# B&R Automation Studio project OpcUaSample410_BrbLibUa103 (part 6)

#### BrbStringPadLeft.c - Füllt einen String auf der linken Seite mit einem Füllzeichen auf eine bestimme Länge
```c
/********************************************************************
 * COPYRIGHT -- Bernecker + Rainer
 ********************************************************************
 * Library: BrbLib
 * File: BrbStringPadLeft.c
 * Author: niedermeierr
 * Created: June 11, 2013
 ********************************************************************
 * Implementation of library BrbLib
 ********************************************************************/

#include <bur/plctypes.h>
#ifdef __cplusplus
	extern "C"
	{
#endif

#include "BrbLib.h"
#include <string.h>

#ifdef __cplusplus
	};
#endif

// NOLINTBEGIN(readability-*, bugprone-easily-swappable-parameters, clang-diagnostic-invalid-utf8, clang-diagnostic-invalid-source-encoding, clang-diagnostic-pointer-arith, clang-diagnostic-strict-prototypes, hicpp-uppercase-literal-suffix, cppcoreguidelines-*, performance-*)

/* Füllt einen String auf der linken Seite mit einem Füllzeichen auf eine bestimme Länge */
plcbit BrbStringPadLeft(plcstring* pText, plcstring* pFillChar, unsigned long nLen)
{
	BOOL bResult = 0;
	UDINT nTextLen = strlen(pText);
	DINT nFillLen = (DINT)nLen - (DINT)nTextLen;
	USINT* pChar = (USINT*)pText;
	if(nFillLen > 0)
	{
		// Text nach rechts schieben
		memmove(pText+nFillLen, pText, nTextLen+1);
		// Füllzeichen einsetzen
		while(pChar < (USINT*)(pText+nFillLen))
		{
			*pChar = (USINT)*pFillChar;
			pChar++;
		}
		bResult = 1;
	}
	return bResult;
}

// NOLINTEND(readability-*, bugprone-easily-swappable-parameters, clang-diagnostic-invalid-utf8, clang-diagnostic-invalid-source-encoding, clang-diagnostic-pointer-arith, clang-diagnostic-strict-prototypes, hicpp-uppercase-literal-suffix, cppcoreguidelines-*, performance-*)
```

#### BrbStringPadRight.c - Füllt einen String auf der rechten Seite mit einem Füllzeichen auf eine bestimme Länge
```c
/********************************************************************
 * COPYRIGHT -- Bernecker + Rainer
 ********************************************************************
 * Library: BrbLib
 * File: BrbStringPadRight.c
 * Author: niedermeierr
 * Created: June 11, 2013
 ********************************************************************
 * Implementation of library BrbLib
 ********************************************************************/

#include <bur/plctypes.h>
#ifdef __cplusplus
	extern "C"
	{
#endif

#include "BrbLib.h"
#include <string.h>

#ifdef __cplusplus
	};
#endif

// NOLINTBEGIN(readability-*, bugprone-easily-swappable-parameters, clang-diagnostic-invalid-utf8, clang-diagnostic-invalid-source-encoding, clang-diagnostic-pointer-arith, clang-diagnostic-strict-prototypes, hicpp-uppercase-literal-suffix, cppcoreguidelines-*, performance-*)

/* Füllt einen String auf der rechten Seite mit einem Füllzeichen auf eine bestimme Länge */
plcbit BrbStringPadRight(plcstring* pText, plcstring* pFillChar, unsigned long nLen)
{
	BOOL bResult = 0;
	UDINT nTextLen = strlen(pText);
	DINT nFillLen = (DINT)nLen - (DINT)nTextLen;
	USINT* pChar = (USINT*)pText + nTextLen;
	if(nFillLen > 0)
	{
		// Füllzeichen einsetzen
		while(pChar < (USINT*)(pText+nLen))
		{
			*pChar = (USINT)*pFillChar;
			pChar++;
		}
		bResult = 1;
	}
	// Terminierung
	*pChar = 0;
	return bResult;
}

// NOLINTEND(readability-*, bugprone-easily-swappable-parameters, clang-diagnostic-invalid-utf8, clang-diagnostic-invalid-source-encoding, clang-diagnostic-pointer-arith, clang-diagnostic-strict-prototypes, hicpp-uppercase-literal-suffix, cppcoreguidelines-*, performance-*)
```

#### BrbStringTrimLeft.c - Schneidet eine Zeichenfolge auf der linken Seite eines Textes heraus
```c
/********************************************************************
 * COPYRIGHT -- Bernecker + Rainer
 ********************************************************************
 * Library: BrbLib
 * File: BrbStringTrimLeft.c
 * Author: niedermeierr
 * Created: December 03, 2013
 ********************************************************************
 * Implementation of library BrbLib
 ********************************************************************/

#include <bur/plctypes.h>
#ifdef __cplusplus
	extern "C"
	{
#endif

#include "BrbLib.h"
#include <string.h>

#ifdef __cplusplus
	};
#endif

// NOLINTBEGIN(readability-*, bugprone-easily-swappable-parameters, clang-diagnostic-invalid-utf8, clang-diagnostic-invalid-source-encoding, clang-diagnostic-pointer-arith, clang-diagnostic-strict-prototypes, hicpp-uppercase-literal-suffix, cppcoreguidelines-*, performance-*)

/* Schneidet eine Zeichenfolge auf der linken Seite eines Textes heraus */
plcbit BrbStringTrimLeft(plcstring* pText, plcstring* pTrim)
{
	BOOL bResult = 0;
	UDINT nTrimLen = strlen(pTrim);
	BOOL bLeave = 0;
	do
	{
		if(BrbStringStartsWith(pText, pTrim) == 1)
		{
			BrbStringCut(pText, 0, nTrimLen, 0);
			bResult = 1;
		}
		else
		{
			bLeave = 1;
		}
	} while(bLeave == 0);
	return bResult;
}

// NOLINTEND(readability-*, bugprone-easily-swappable-parameters, clang-diagnostic-invalid-utf8, clang-diagnostic-invalid-source-encoding, clang-diagnostic-pointer-arith, clang-diagnostic-strict-prototypes, hicpp-uppercase-literal-suffix, cppcoreguidelines-*, performance-*)
```

#### BrbStringTrimRight.c - Schneidet eine Zeichenfolge auf der rechten Seite eines Textes heraus
```c
/********************************************************************
 * COPYRIGHT -- Bernecker + Rainer
 ********************************************************************
 * Library: BrbLib
 * File: BrbStringTrimRight.c
 * Author: niedermeierr
 * Created: December 03, 2013
 ********************************************************************
 * Implementation of library BrbLib
 ********************************************************************/

#include <bur/plctypes.h>
#ifdef __cplusplus
	extern "C"
	{
#endif

#include "BrbLib.h"
#include <string.h>

#ifdef __cplusplus
	};
#endif

// NOLINTBEGIN(readability-*, bugprone-easily-swappable-parameters, clang-diagnostic-invalid-utf8, clang-diagnostic-invalid-source-encoding, clang-diagnostic-pointer-arith, clang-diagnostic-strict-prototypes, hicpp-uppercase-literal-suffix, cppcoreguidelines-*, performance-*)

/* Schneidet eine Zeichenfolge auf der rechten Seite eines Textes heraus */
plcbit BrbStringTrimRight(plcstring* pText, plcstring* pTrim)
{
	BOOL bResult = 0;
	UDINT nTrimLen = strlen(pTrim);
	BOOL bLeave = 0;
	do
	{
		if(BrbStringEndsWith(pText, pTrim) == 1)
		{
			UDINT nTextLen = strlen(pText);
			BrbStringCut(pText, nTextLen-nTrimLen, nTrimLen, 0);
			bResult = 1;
		}
		else
		{
			bLeave = 1;
		}
	} while(bLeave == 0);
	return bResult;
}

// NOLINTEND(readability-*, bugprone-easily-swappable-parameters, clang-diagnostic-invalid-utf8, clang-diagnostic-invalid-source-encoding, clang-diagnostic-pointer-arith, clang-diagnostic-strict-prototypes, hicpp-uppercase-literal-suffix, cppcoreguidelines-*, performance-*)
```

#### BrbStringSplit.c - Spaltet einen Text in mehrere String aufgrund eines Trennzeichens
```c
/********************************************************************
 * COPYRIGHT -- Bernecker + Rainer
 ********************************************************************
 * Library: BrbLib
 * File: BrbStringSplit.c
 * Author: niedermeierr
 * Created: June 17, 2013
 ********************************************************************
 * Implementation of library BrbLib
 ********************************************************************/

#include <bur/plctypes.h>
#ifdef __cplusplus
	extern "C"
	{
#endif

#include "BrbLib.h"
#include <string.h>

#ifdef __cplusplus
	};
#endif

// NOLINTBEGIN(readability-*, bugprone-easily-swappable-parameters, clang-diagnostic-invalid-utf8, clang-diagnostic-invalid-source-encoding, clang-diagnostic-pointer-arith, clang-diagnostic-strict-prototypes, hicpp-uppercase-literal-suffix, cppcoreguidelines-*, performance-*)

/* Spaltet einen Text in mehrere Strings aufgrund eines Trennzeichens */
unsigned long BrbStringSplit(plcstring* pText, plcstring* pSep, unsigned long pSplitArray, unsigned long nArrayIndexMax, unsigned long nEntrySize)
{
	if(nEntrySize <= 1)
	{
		// String-Grösse zu klein
		return 0;
	}
	UDINT nResult = 0;
	UDINT nLenText = strlen(pText);
	UDINT nLenSep = strlen(pSep);
	// Der Einfachkeit halber wird das Array in einer MemList verwaltet
	BrbMemListManagement_Typ ListMan;
	ListMan.pList = pSplitArray;
	ListMan.nIndexMax = nArrayIndexMax;
	ListMan.nEntryLength = nEntrySize;
	BrbMemListClear(&ListMan);
	// Text von vorne nach hinten nach Trennzeichen durchsuchen
	STRING* pEntryTextStart = pText;
	STRING* pEntryTextEnd = 0;
	UDINT nCharIndex = 0;
	do
	{
		// Trennzeichen vergleichen
		if((memcmp((pText + nCharIndex), pSep, nLenSep) == 0) || nCharIndex == nLenText-1)
		{
			// Trennzeichen gefunden -> Splittext holen und in Array eintragen
			if(nCharIndex == nLenText-1)
			{
				// Kein Trennzeichen am Ende
				pEntryTextEnd = pText + nCharIndex + 1;
			}
			else
			{
				pEntryTextEnd = pText + nCharIndex;
			}
			STRING sEntryText[nEntrySize];
			memset(sEntryText, 0, sizeof(sEntryText));
			DINT nNeededEntrySize = (DINT)pEntryTextEnd - (DINT)pEntryTextStart + 1;
			if((DINT)nEntrySize < nNeededEntrySize)
			{
				pEntryTextEnd = pEntryTextStart + nEntrySize - 1;
			}
			BrbStringGetSubTextByAdr(pEntryTextStart, pEntryTextEnd, sEntryText);
			if(strlen(sEntryText) > 0 && strcmp(sEntryText, pSep) != 0)
			{
				BrbMemListIn(&ListMan, ListMan.nEntryCount, (UDINT)&sEntryText);
				nResult += 1;
			}
			// Weitermachen mit Text nach Trennzeichen
			nCharIndex += nLenSep;
			pEntryTextStart = pText + nCharIndex;
		}
		else
		{
			nCharIndex += 1;
		}
	} while(nCharIndex<nLenText);
	return nResult;
}

// NOLINTEND(readability-*, bugprone-easily-swappable-parameters, clang-diagnostic-invalid-utf8, clang-diagnostic-invalid-source-encoding, clang-diagnostic-pointer-arith, clang-diagnostic-strict-prototypes, hicpp-uppercase-literal-suffix, cppcoreguidelines-*, performance-*)
```

#### BrbStringSplitEmpty.c - Spaltet einen Text in mehrere String aufgrund eines Trennzeichens
```c
/********************************************************************
 * COPYRIGHT -- Bernecker + Rainer
 ********************************************************************
 * Library: BrbLib
 * File: BrbStringSplitEmpty.c
 * Author: niedermeierr
 * Created: May 17, 2021
 ********************************************************************
 * Implementation of library BrbLib
 ********************************************************************/

#include <bur/plctypes.h>
#ifdef __cplusplus
	extern "C"
	{
#endif

#include "BrbLib.h"
#include <string.h>

#ifdef __cplusplus
	};
#endif

// NOLINTBEGIN(readability-*, bugprone-easily-swappable-parameters, clang-diagnostic-invalid-utf8, clang-diagnostic-invalid-source-encoding, clang-diagnostic-pointer-arith, clang-diagnostic-strict-prototypes, hicpp-uppercase-literal-suffix, cppcoreguidelines-*, performance-*)

/* Spaltet einen Text in mehrere Strings aufgrund eines Trennzeichens (inkl. Leer-Strings) */
unsigned long BrbStringSplitEmpty(plcstring* pText, plcstring* pSep, unsigned long pSplitArray, unsigned long nArrayIndexMax, unsigned long nEntrySize)
{
	if(nEntrySize <= 1)
	{
		// String-Grösse zu klein
		return 0;
	}
	UDINT nResult = 0;
	UDINT nLenText = strlen(pText);
	UDINT nLenSep = strlen(pSep);
	// Der Einfachkeit halber wird das Array in einer MemList verwaltet
	BrbMemListManagement_Typ ListMan;
	ListMan.pList = pSplitArray;
	ListMan.nIndexMax = nArrayIndexMax;
	ListMan.nEntryLength = nEntrySize;
	BrbMemListClear(&ListMan);
	// Text von vorne nach hinten nach Trennzeichen durchsuchen
	STRING* pEntryTextStart = pText;
	STRING* pEntryTextEnd = 0;
	UDINT nCharIndex = 0;
	do
	{
		// Trennzeichen vergleichen
		if((memcmp((pText + nCharIndex), pSep, nLenSep) == 0) || nCharIndex == nLenText-1)
		{
			// Trennzeichen gefunden -> Splittext holen und in Array eintragen
			if((memcmp((pText + nCharIndex), pSep, nLenSep) != 0) && nCharIndex == nLenText-1)
			{
				// Kein Trennzeichen am Ende
				pEntryTextEnd = pText + nCharIndex + 1;
			}
			else
			{
				pEntryTextEnd = pText + nCharIndex;
			}
			STRING sEntryText[nEntrySize];
			memset(sEntryText, 0, sizeof(sEntryText));
			DINT nNeededEntrySize = (DINT)pEntryTextEnd - (DINT)pEntryTextStart + 1;
			if((DINT)nEntrySize < nNeededEntrySize)
			{
				pEntryTextEnd = pEntryTextStart + nEntrySize - 1;
			}
			BrbStringGetSubTextByAdr(pEntryTextStart, pEntryTextEnd, sEntryText);
			if(strcmp(sEntryText, pSep) == 0)
			{
				memset(sEntryText, 0, sizeof(sEntryText));
			}
			BrbMemListIn(&ListMan, ListMan.nEntryCount, (UDINT)&sEntryText);
			nResult += 1;
			// Weitermachen mit Text nach Trennzeichen
			nCharIndex += nLenSep;
			pEntryTextStart = pText + nCharIndex;
		}
		else
		{
			nCharIndex += 1;
		}
	} while(nCharIndex<nLenText);
	if(pEntryTextEnd != 0)
	{
		if(BrbStringEndsWith(pEntryTextEnd, pSep) == 1)
		{
			// Text endet mit Trennzeichen -> noch einen leeren Eintrag hinzufügen
			STRING sEntryText[nEntrySize];
			memset(sEntryText, 0, sizeof(sEntryText));
			BrbMemListIn(&ListMan, ListMan.nEntryCount, (UDINT)&sEntryText);
			nResult += 1;
		}
	}
	return nResult;
}

// NOLINTEND(readability-*, bugprone-easily-swappable-parameters, clang-diagnostic-invalid-utf8, clang-diagnostic-invalid-source-encoding, clang-diagnostic-pointer-arith, clang-diagnostic-strict-prototypes, hicpp-uppercase-literal-suffix, cppcoreguidelines-*, performance-*)
```

#### BrbStringConvertRealFromExp.c - Konvertiert eine exponentielle Notation in einen Real-Wert
```c
/********************************************************************
 * COPYRIGHT -- Bernecker + Rainer
 ********************************************************************
 * Library: BrbLib
 * File: BrbStringConvertRealFromExp.c
 * Author: niedermeierr
 * Created: December 03, 2013
 ********************************************************************
 * Implementation of library BrbLib
 ********************************************************************/

#include <bur/plctypes.h>
#ifdef __cplusplus
	extern "C"
	{
#endif

#include "BrbLib.h"
#include <string.h>
#include <AnsiCFunc.h>

#ifdef __cplusplus
	};
#endif

// NOLINTBEGIN(readability-*, bugprone-easily-swappable-parameters, clang-diagnostic-invalid-utf8, clang-diagnostic-invalid-source-encoding, clang-diagnostic-pointer-arith, clang-diagnostic-strict-prototypes, hicpp-uppercase-literal-suffix, cppcoreguidelines-*, performance-*)

/* Konvertiert eine exponentielle Notation in einen Real-Wert */
unsigned short BrbStringConvertRealFromExp(plcstring* pValue, plcstring* pResult, unsigned long nResultSize) // NOLINT(readability-function-cognitive-complexity)
{
	memset(pResult, 0, nResultSize);
	UDINT nValueLen = strlen(pValue);
	STRING* pExpStart = BrbStringGetAdrOf(pValue, "e", nValueLen);
	if(pExpStart > pValue)
	{
		// "e" enthalten -> Zahl vor dem "e"
		STRING sReal[50];
		memset(sReal, 0, sizeof(sReal));
		BrbStringGetSubTextByAdr(pValue, pExpStart, sReal); // NOLINT(readability-suspicious-call-argument)
		// Vorzeichen, Anzahl der Vorkomma-Stellen, Stelle des Kommas und Anzahl der Nachkomma-Stellen
		BOOL bMinus = 0;
		// Vorzeichen löschen
		BrbStringTrimLeft(sReal, "+");
		if(BrbStringStartsWith(sReal, "-") == 1)
		{
			bMinus = 1;
			BrbStringTrimLeft(sReal, "-");
		}
		// Führende Nullen löschen
		BrbStringTrimLeft(sReal, "0");

		STRING* pRealDot = BrbStringGetAdrOf(sReal, ".", nValueLen);
		UDINT nIntegerDigits = 0;
		DINT nDotDigit = 0;
		UDINT nFractionDigits = 0;
		if((UDINT)pRealDot >= (UDINT)&sReal)
		{
			// Punkt enthalten
			// Folgende Nullen nach dem Punkt löschen
			BrbStringTrimRight(sReal, "0");
			if(BrbStringEndsWith(sReal, ".") == 1)
			{
				brsstrcat((UDINT)&sReal, (UDINT)&"0");
			}
			UDINT nRealLen = strlen(sReal);
			nIntegerDigits = (UDINT)pRealDot - (UDINT)sReal;
			nDotDigit = (DINT)((UDINT)pRealDot - (UDINT)&sReal);
			nFractionDigits = (UDINT)&sReal + nRealLen - (UDINT)pRealDot - 1;
			// Punkt löschen
			BrbStringReplace(sReal, ".", "");
		}
		else
		{
			// Punkt nicht enthalten
			nIntegerDigits = (UDINT)pExpStart - (UDINT)pValue;
			nDotDigit = -1;
			nFractionDigits = 0;
		}
		brsstrcpy((UDINT)pResult, (UDINT)&sReal);
		UDINT nExpLen = strlen(pExpStart);
		if(nExpLen > 1)
		{
			// Zahl nach dem "e"
			STRING sExp[50];
			memset(sExp, 0, sizeof(sExp));
			BrbStringGetSubTextByLen(pExpStart + 1, nExpLen - 1, sExp);
			DINT nExp = brsatoi((UDINT)&sExp);
			// Vorzeichen des Exponenten
			STRING* pExpMinus = BrbStringGetAdrOf(pExpStart, "-", nExpLen);
			if(pExpMinus > pExpStart && nExp != 0)
			{
				// Exponent ist negativ -> Nullen voranstellen
				UDINT nAddZero = (UDINT)((DINT)abs(nExp) - (DINT)nIntegerDigits) + 1;
				UDINT nCount = 0;
				for(nCount=0; nCount<nAddZero; nCount++)
				{
					BrbStringInsert(pResult, 0, "0");
				}
				// Punkt einfügen
				BrbStringInsert(pResult, 1, ".");
			}
			else
			{
				// Exponent ist positiv
				if((DINT)nFractionDigits <= nExp)
				{
					// Nullen anhängen
					UDINT nAddZero = (UDINT)(nExp - (DINT)nFractionDigits);
					UDINT nCount = 0;
					for(nCount=0; nCount<nAddZero; nCount++)
					{
						brsstrcat((UDINT)pResult, (UDINT)&"0");
					}
				}
				else
				{
					// Punkt einfügen
					if(nDotDigit > -1)
					{
						UDINT nIndex = (UDINT)(nDotDigit + nExp);
						BrbStringInsert(pResult, nIndex, ".");
					}
				}
			}
			// Führende Nullen löschen
			BrbStringTrimLeft(pResult, "0");
			// Null vor dem Punkt wieder einfügen
			if(BrbStringStartsWith(pResult, ".") == 1)
			{
				BrbStringInsert(pResult, 0, "0");
			}
			// Vorzeichen einfügen
			if(bMinus == 1)
			{
				BrbStringInsert(pResult, 0, "-");
			}
		}
	}
	else
	{
		// "e" nicht enthalten
		brsstrcpy((UDINT)pResult, (UDINT)pValue);
		// Vorzeichen löschen
		BrbStringTrimLeft(pResult, "+");
		BOOL bMinus = 0;
		if(BrbStringStartsWith(pResult, "-") == 1)
		{
			bMinus = 1;
			BrbStringTrimLeft(pResult, "-");
		}
		// Führende Nullen löschen
		BrbStringTrimLeft(pResult, "0");
		// Null vor dem Punkt wieder einfügen
		if(BrbStringStartsWith(pResult, ".") == 1)
		{
			BrbStringInsert(pResult, 0, "0");
		}
		// Folgende Nullen nach dem Punkt löschen
		UDINT nLen = strlen(pResult);
		STRING* pDot = BrbStringGetAdrOf(pResult, ".", nLen);
		if(pDot > pResult)
		{
			BrbStringTrimRight(pResult, "0");
			if(BrbStringEndsWith(pResult, ".") == 1)
			{
				brsstrcat((UDINT)pResult, (UDINT)&"0");
			}
		}
		if(strlen(pResult) == 0)
		{
			brsstrcat((UDINT)pResult, (UDINT)&"0.0");
		}
		// Vorzeichen einfügen
		if(bMinus == 1)
		{
			BrbStringInsert(pResult, 0, "-");
		}
	}
	return eBRB_ERR_OK;
}

// NOLINTEND(readability-*, bugprone-easily-swappable-parameters, clang-diagnostic-invalid-utf8, clang-diagnostic-invalid-source-encoding, clang-diagnostic-pointer-arith, clang-diagnostic-strict-prototypes, hicpp-uppercase-literal-suffix, cppcoreguidelines-*, performance-*)
```

#### BrbStringConvertRealToExp.c - Konvertiert einen Real-Wert in eine exponentielle Notation
```c
/********************************************************************
 * COPYRIGHT -- Bernecker + Rainer
 ********************************************************************
 * Library: BrbLib
 * File: BrbStringConvertRealToExp.c
 * Author: niedermeierr
 * Created: December 03, 2013
 ********************************************************************
 * Implementation of library BrbLib
 ********************************************************************/

#include <bur/plctypes.h>
#ifdef __cplusplus
	extern "C"
	{
#endif

#include "BrbLib.h"
#include <string.h>
#include <AnsiCFunc.h>

#ifdef __cplusplus
	};
#endif

// NOLINTBEGIN(readability-*, bugprone-easily-swappable-parameters, clang-diagnostic-invalid-utf8, clang-diagnostic-invalid-source-encoding, clang-diagnostic-pointer-arith, clang-diagnostic-strict-prototypes, hicpp-uppercase-literal-suffix, cppcoreguidelines-*, performance-*)

/* Konvertiert einen Real-Wert in eine exponentielle Notation */
unsigned short BrbStringConvertRealToExp(plcstring* pValue, plcstring* pResult, unsigned long nResultSize) // NOLINT(readability-function-cognitive-complexity)
{
	memset(pResult, 0, nResultSize);
	UDINT nValueLen = strlen(pValue);
	STRING* pExpStart = BrbStringGetAdrOf(pValue, "e", nValueLen);
	if(pExpStart == 0)
	{
		// "e" nicht enthalten
		brsstrcpy((UDINT)pResult, (UDINT)pValue);
		// Vorzeichen löschen
		BrbStringTrimLeft(pResult, "+");
		BOOL bMinus = 0;
		if(BrbStringStartsWith(pResult, "-") == 1)
		{
			bMinus = 1;
			BrbStringTrimLeft(pResult, "-");
		}
		// Führende Nullen löschen
		BrbStringTrimLeft(pResult, "0");
		// Null vor dem Punkt wieder einfügen
		if(BrbStringStartsWith(pResult, ".") == 1)
		{
			BrbStringInsert(pResult, 0, "0");
		}
		else if(brsstrlen((UDINT)pResult) == 0)
		{
			brsstrcat((UDINT)pResult, (UDINT)&"0.0");
		}
		// Folgende Nullen nach dem Punkt löschen
		UDINT nLen = strlen(pResult);
		STRING* pDot = BrbStringGetAdrOf(pResult, ".", nLen);
		if(pDot > pResult)
		{
			BrbStringTrimRight(pResult, "0");
			if(BrbStringEndsWith(pResult, ".") == 1)
			{
				brsstrcat((UDINT)pResult, (UDINT)&"0");
			}
			nLen = strlen(pResult);
			pDot = BrbStringGetAdrOf(pResult, ".", nLen);
		}
		// Vorzeichen des Exponenten feststellen
		BOOL bExpMinus = 0;
		if(BrbStringStartsWith(pResult, "0") == 1)
		{
			// 0.0012345
			// Erstes Zeichen ist "0" -> Exponent negativ
			bExpMinus = 1;
		}
		else
		{
			// 123.45
			// Erstes Zeichen ist keine "0" -> Exponent positiv
			bExpMinus = 0;
		}
		// Exponent feststellen
		DINT nExp = 0;
		if(bExpMinus == 1)
		{
			// Negativer Exponent
			if(pDot > pResult)
			{
				// Punkt enthalten
				nExp = 1;
				USINT* pChar = 0;
				USINT* pEnd =(USINT*)pResult + nLen - 1;
				// Anzahl der Nullen vom Punkt bis zur ersten relevanten Ziffer
				for(pChar=(USINT*)pDot+1; pChar<=pEnd; pChar++)
				{
					if(*pChar == 48)
					{
						nExp += 1;
					}
					else
					{
						break;
					}
				}
				UDINT nDotDigit = (UDINT)pDot - (UDINT)pResult;
				UDINT nCutLen = nDotDigit + (UDINT)nExp;
				// Alle Zeichen bis zur ersten relevanten Ziffer löschen
				BrbStringCut(pResult, 0, nCutLen, 0);
			}
			else
			{
				// Punkt nicht enthalten
				nExp = 0;
			}
		}
		else
		{
			// Positiver Exponent
			if(pDot > pResult)
			{
				// Punkt enthalten
				DINT nDotDigit = (DINT)((UDINT)pDot - (UDINT)pResult);
				nExp = nDotDigit - 1;
				// Punkt löschen
				BrbStringReplace(pResult, ".", "");
			}
			else
			{
				// Punkt nicht enthalten
				nExp = (DINT)nLen - 1;
			}
		}
		if(brsstrlen((UDINT)pResult) == 0)
		{
			brsstrcat((UDINT)pResult, (UDINT)&"0.0e+000");
		}
		else
		{
			// Punkt an 2. Stelle einfügen (1 Vorkomma-Stelle)
			BrbStringInsert(pResult, 1, ".");
			// Folgende Nullen löschen
			BrbStringTrimRight(pResult, "0");
			// "e" anhängen
			brsstrcat((UDINT)pResult, (UDINT)&"e");
			// Exponent-Vorzeichen
			if(bExpMinus == 0)
			{
				brsstrcat((UDINT)pResult, (UDINT)&"+");
			}
			else
			{
				brsstrcat((UDINT)pResult, (UDINT)&"-");
			}
			// Exponent mit mindestens 3 Stellen anhängen
			STRING sExp[50];
			brsitoa(nExp, (UDINT)&sExp);
			BrbStringPadLeft(sExp, "0", 3);
			brsstrcat((UDINT)pResult, (UDINT)&sExp);
			// Vorzeichen einfügen
			if(bMinus == 1)
			{
				BrbStringInsert(pResult, 0, "-");
			}
		}
	}
	else
	{
		// "e" enthalten
		STRING sTemp[nResultSize];
		BrbStringConvertRealFromExp(pValue, sTemp, sizeof(sTemp));
		BrbStringConvertRealToExp(sTemp, pResult, nResultSize);
	}
	return eBRB_ERR_OK;
}

// NOLINTEND(readability-*, bugprone-easily-swappable-parameters, clang-diagnostic-invalid-utf8, clang-diagnostic-invalid-source-encoding, clang-diagnostic-pointer-arith, clang-diagnostic-strict-prototypes, hicpp-uppercase-literal-suffix, cppcoreguidelines-*, performance-*)
```

#### BrbStringFormatFractionDigits.c - Formatiert einen String-Wert auf Nachkommastellen
```c
/********************************************************************
 * COPYRIGHT -- Bernecker + Rainer
 ********************************************************************
 * Library: BrbLib
 * File: BrbStringFormatFractionDigits.c
 * Author: niedermeierr
 * Created: June 11, 2013
 ********************************************************************
 * Implementation of library BrbLib
 ********************************************************************/

#include <bur/plctypes.h>
#ifdef __cplusplus
	extern "C"
	{
#endif

#include "BrbLib.h"
#include <string.h>

#ifdef __cplusplus
	};
#endif

// NOLINTBEGIN(readability-*, bugprone-easily-swappable-parameters, clang-diagnostic-invalid-utf8, clang-diagnostic-invalid-source-encoding, clang-diagnostic-pointer-arith, clang-diagnostic-strict-prototypes, hicpp-uppercase-literal-suffix, cppcoreguidelines-*, performance-*)

/* Formatiert einen Real-String-Wert auf Nachkommastellen */
unsigned short  BrbStringFormatFractionDigits(plcstring* pValue, unsigned long nValueSize, unsigned short nFractionsDigits)
{
	STRING sTemp[nValueSize+1];
	BrbStringConvertRealFromExp(pValue, sTemp, sizeof(sTemp));
	brsstrcpy((UDINT)pValue, (UDINT)&sTemp);
	UDINT nValueLen = strlen(pValue);
	STRING* pDot = BrbStringGetAdrOf(pValue, ".", nValueLen);
	if(pDot > pValue)
	{
		// Punkt gefunden
		UDINT nLenAfterDot = ((UDINT)pValue + nValueLen) - (UDINT)pDot - 1;
		if(nLenAfterDot > nFractionsDigits)
		{
			if(nFractionsDigits > 0)
			{
				*(pDot + nFractionsDigits + 1) = 0;
			}
			else
			{
				*pDot = 0;
			}
		}
		else if(nLenAfterDot < nFractionsDigits)
		{
			UDINT nMissingDigits = nFractionsDigits - nLenAfterDot;
			UDINT nMissingChars = 0;
			for(nMissingChars=0; nMissingChars<nMissingDigits; nMissingChars++)
			{
				BrbStringCat(pValue, "0", nValueSize);
			}
		}
	}
	else
	{
		// Punkt nicht gefunden
		if(nFractionsDigits > 0)
		{
			BrbStringCat(pValue, ".", nValueSize);
			UDINT nMissingChars = 0;
			for(nMissingChars=0; nMissingChars<nFractionsDigits; nMissingChars++)
			{
				BrbStringCat(pValue, "0", nValueSize);
			}
		}
	}
	return eBRB_ERR_OK;
}

// NOLINTEND(readability-*, bugprone-easily-swappable-parameters, clang-diagnostic-invalid-utf8, clang-diagnostic-invalid-source-encoding, clang-diagnostic-pointer-arith, clang-diagnostic-strict-prototypes, hicpp-uppercase-literal-suffix, cppcoreguidelines-*, performance-*)
```

#### BrbStringSwap.c - Dreht die Reihenfolge der Zeichen in einem Text
```c
/********************************************************************
 * COPYRIGHT -- Bernecker + Rainer
 ********************************************************************
 * Library: BrbLib
 * File: BrbStringSwap.c
 * Author: niedermeierr
 * Created: June 11, 2013
 ********************************************************************
 * Implementation of library BrbLib
 ********************************************************************/

#include <bur/plctypes.h>
#ifdef __cplusplus
	extern "C"
	{
#endif

#include "BrbLib.h"
#include <string.h>

#ifdef __cplusplus
	};
#endif

// NOLINTBEGIN(readability-*, bugprone-easily-swappable-parameters, clang-diagnostic-invalid-utf8, clang-diagnostic-invalid-source-encoding, clang-diagnostic-pointer-arith, clang-diagnostic-strict-prototypes, hicpp-uppercase-literal-suffix, cppcoreguidelines-*, performance-*)

/* Dreht die Reihenfolge der Zeichen in einem Text */
plcbit BrbStringSwap(plcstring* pText, plcstring* pSwapped, unsigned long nSwappedSize)
{
	BOOL bResult = 0;
	memset(pSwapped, 0, nSwappedSize);
	UDINT nIndex = 0;
	USINT* pCharText = 0;
	USINT* pCharSwapped = 0;
	UDINT nTextLen = strlen(pText);
	if(nTextLen <= nSwappedSize)
	{
		for(nIndex=0; nIndex<nTextLen; nIndex++)
		{
			pCharText = (USINT*)(pText + nIndex);
			pCharSwapped = (USINT*)(pSwapped + nTextLen - nIndex - 1);
			*pCharSwapped = *pCharText;
		}
		bResult = 1;
	}
	return bResult;
}

// NOLINTEND(readability-*, bugprone-easily-swappable-parameters, clang-diagnostic-invalid-utf8, clang-diagnostic-invalid-source-encoding, clang-diagnostic-pointer-arith, clang-diagnostic-strict-prototypes, hicpp-uppercase-literal-suffix, cppcoreguidelines-*, performance-*)
```

#### BrbStringToUpper.c - Konvertiert einen String zu Großbuchstaben
```c
/********************************************************************
 * COPYRIGHT -- Bernecker + Rainer
 ********************************************************************
 * Library: BrbLib
 * File: BrbStringToUpper.c
 * Author: niedermeierr
 * Created: March 04, 2015
 ********************************************************************
 * Implementation of library BrbLib
 ********************************************************************/

#include <bur/plctypes.h>
#ifdef __cplusplus
	extern "C"
	{
#endif

#include "BrbLib.h"
#include <string.h>

#ifdef __cplusplus
	};
#endif

// NOLINTBEGIN(readability-*, bugprone-easily-swappable-parameters, clang-diagnostic-invalid-utf8, clang-diagnostic-invalid-source-encoding, clang-diagnostic-pointer-arith, clang-diagnostic-strict-prototypes, hicpp-uppercase-literal-suffix, cppcoreguidelines-*, performance-*)

/* Konvertiert einen String zu Großbuchstaben */
plcbit BrbStringToUpper(plcstring* pText)
{
	BOOL bResult = 0;
	UDINT nTextLen = strlen(pText);
	UDINT nIndex = 0;
	USINT* pChar = 0;
	for(nIndex=0; nIndex<nTextLen; nIndex++)
	{
		pChar = (USINT*)(pText + nIndex);
		if(*pChar >= 97 && *pChar <= 122)
		{
			*pChar = *pChar - 32;
			bResult = 1;
		}
	}
	return bResult;
}

// NOLINTEND(readability-*, bugprone-easily-swappable-parameters, clang-diagnostic-invalid-utf8, clang-diagnostic-invalid-source-encoding, clang-diagnostic-pointer-arith, clang-diagnostic-strict-prototypes, hicpp-uppercase-literal-suffix, cppcoreguidelines-*, performance-*)
```

#### BrbStringToLower.c - Konvertiert einen String zu Kleinbuchstaben
```c
/********************************************************************
 * COPYRIGHT -- Bernecker + Rainer
 ********************************************************************
 * Library: BrbLib
 * File: BrbStringToLower.c
 * Author: niedermeierr
 * Created: March 04, 2015
 ********************************************************************
 * Implementation of library BrbLib
 ********************************************************************/

#include <bur/plctypes.h>
#ifdef __cplusplus
	extern "C"
	{
#endif

#include "BrbLib.h"
#include <string.h>

#ifdef __cplusplus
	};
#endif

// NOLINTBEGIN(readability-*, bugprone-easily-swappable-parameters, clang-diagnostic-invalid-utf8, clang-diagnostic-invalid-source-encoding, clang-diagnostic-pointer-arith, clang-diagnostic-strict-prototypes, hicpp-uppercase-literal-suffix, cppcoreguidelines-*, performance-*)

/* Konvertiert einen String zu Kleinbuchstaben */
plcbit BrbStringToLower(plcstring* pText)
{
	BOOL bResult = 0;
	UDINT nTextLen = strlen(pText);
	UDINT nIndex = 0;
	USINT* pChar = 0;
	for(nIndex=0; nIndex<nTextLen; nIndex++)
	{
		pChar = (USINT*)(pText + nIndex);
		if(*pChar >= 65 && *pChar <= 90)
		{
			*pChar = *pChar + 32;
			bResult = 1;
		}
	}
	return bResult;
}

// NOLINTEND(readability-*, bugprone-easily-swappable-parameters, clang-diagnostic-invalid-utf8, clang-diagnostic-invalid-source-encoding, clang-diagnostic-pointer-arith, clang-diagnostic-strict-prototypes, hicpp-uppercase-literal-suffix, cppcoreguidelines-*, performance-*)
```

#### BrbStringIsNumerical.c - Gibt zurück, ob ein Text eine Nummer enthält
```c
/********************************************************************
 * COPYRIGHT -- Bernecker + Rainer
 ********************************************************************
 * Library: BrbLib
 * File: BrbStringIsNumerical.c
 * Author: niedermeierr
 * Created: March 18, 2015
 ********************************************************************
 * Implementation of library BrbLib
 ********************************************************************/

#include <bur/plctypes.h>
#ifdef __cplusplus
	extern "C"
	{
#endif

#include "BrbLib.h"
#include <string.h>

#ifdef __cplusplus
	};
#endif

// NOLINTBEGIN(readability-*, bugprone-easily-swappable-parameters, clang-diagnostic-invalid-utf8, clang-diagnostic-invalid-source-encoding, clang-diagnostic-pointer-arith, clang-diagnostic-strict-prototypes, hicpp-uppercase-literal-suffix, cppcoreguidelines-*, performance-*)

/* Gibt zurück, ob ein Text eine Nummer enthält */
plcbit BrbStringIsNumerical(plcstring* pText) // NOLINT(readability-function-cognitive-complexity)
{
	BOOL bResult = 1;
	UDINT nTextLen = strlen(pText);
	if(nTextLen == 0)
	{
		bResult = 0;
	}
	else
	{
		UDINT nIndex = 0;
		USINT* pChar = 0;
		UINT nCountSeparator = 0;
		DINT nIndexExp = -1;
		for(nIndex=0; nIndex<nTextLen; nIndex++)
		{
			pChar = (USINT*)(pText + nIndex);
			// NOLINTBEGIN(bugprone-branch-clone)
			if(*pChar == 43)
			{
				// Plus
				if(nIndex != 0 && nIndexExp != (DINT)nIndex-1)
				{
					// Nicht am Anfang oder nach "e"
					bResult = 0;
					break;
				}
			}
			else if(*pChar == 45)
			{
				// Minus
				if(nIndex != 0 && nIndexExp != (DINT)nIndex-1)
				{
					// Nicht am Anfang oder nach "e"
					bResult = 0;
					break;
				}
			}
			else if(*pChar == 44)
			{
				// Komma
				nCountSeparator++;
				if(nCountSeparator > 1)
				{
					// Mehr als 1 Separartor
					bResult = 0;
					break;
				}
			}
			else if(*pChar == 46)
			{
				// Punkt
				nCountSeparator++;
				if(nCountSeparator > 1)
				{
					// Mehr als 1 Separartor
					bResult = 0;
					break;
				}
			}
			else if(*pChar == 101)
			{
				// e
				if(nIndexExp == -1)
				{
					nIndexExp = (DINT)nIndex;
					if(nIndex >= nTextLen-1)
					{
						// Nach "e" folgt nichts
						bResult = 0;
						break;
					}
				}
				else
				{
					// Zweites "e"
					bResult = 0;
					break;
				}
			}
			else if(!(*pChar >= 48 && *pChar <= 57))
			{
				bResult = 0;
				break;
			}
			// NOLINTEND(bugprone-branch-clone)
		}
	}
	return bResult;
}

// NOLINTEND(readability-*, bugprone-easily-swappable-parameters, clang-diagnostic-invalid-utf8, clang-diagnostic-invalid-source-encoding, clang-diagnostic-pointer-arith, clang-diagnostic-strict-prototypes, hicpp-uppercase-literal-suffix, cppcoreguidelines-*, performance-*)
```

#### BrbStringIsHex.c - Gibt zurück, ob ein Text eine hexadezimale Nummer enthält
```c
/********************************************************************
 * COPYRIGHT -- Bernecker + Rainer
 ********************************************************************
 * Library: BrbLib
 * File: BrbStringIsHex.c
 * Author: niedermeierr
 * Created: January 17, 2017
 ********************************************************************
 * Implementation of library BrbLib
 ********************************************************************/

#include <bur/plctypes.h>
#ifdef __cplusplus
	extern "C"
	{
#endif

#include "BrbLib.h"
#include <string.h>

#ifdef __cplusplus
	};
#endif

// NOLINTBEGIN(readability-*, bugprone-easily-swappable-parameters, clang-diagnostic-invalid-utf8, clang-diagnostic-invalid-source-encoding, clang-diagnostic-pointer-arith, clang-diagnostic-strict-prototypes, hicpp-uppercase-literal-suffix, cppcoreguidelines-*, performance-*)

/* Gibt zurück, ob ein Text eine hexadezimale Nummer enthält */
plcbit BrbStringIsHex(plcstring* pText, plcbit bLowCaseAllowed)
{
	BOOL bResult = 1;
	UDINT nTextLen = strlen(pText);
	if(nTextLen == 0)
	{
		bResult = 0;
	}
	else
	{
		UDINT nIndex = 0;
		USINT* pChar = 0;
		for(nIndex=0; nIndex<nTextLen; nIndex++)
		{
			pChar = (USINT*)(pText + nIndex);
			// NOLINTBEGIN(bugprone-branch-clone)
			if((*pChar >= 48 && *pChar <= 57)) // 0..9
			{
			}
			else if((*pChar >= 65 && *pChar <= 70)) // A..F
			{
			}
			else if((*pChar >= 97 && *pChar <= 102) && bLowCaseAllowed == 1) // a..f
			{
			}
			else
			{
				bResult = 0;
				break;
			}
			// NOLINTEND(bugprone-branch-clone)
		}
	}
	return bResult;
}

// NOLINTEND(readability-*, bugprone-easily-swappable-parameters, clang-diagnostic-invalid-utf8, clang-diagnostic-invalid-source-encoding, clang-diagnostic-pointer-arith, clang-diagnostic-strict-prototypes, hicpp-uppercase-literal-suffix, cppcoreguidelines-*, performance-*)
```

#### BrbStringCountText.c - Zählt das Vorkommen einer Zeichenfolge innerhalb eines Texts
```c
/********************************************************************
 * COPYRIGHT -- Bernecker + Rainer
 ********************************************************************
 * Library: BrbLib
 * File: BrbStringCountText.c
 * Author: niedermeierr
 * Created: April 13, 2016
 ********************************************************************
 * Implementation of library BrbLib
 ********************************************************************/

#include <bur/plctypes.h>
#ifdef __cplusplus
	extern "C"
	{
#endif

#include "BrbLib.h"
#include <string.h>

#ifdef __cplusplus
	};
#endif

// NOLINTBEGIN(readability-*, bugprone-easily-swappable-parameters, clang-diagnostic-invalid-utf8, clang-diagnostic-invalid-source-encoding, clang-diagnostic-pointer-arith, clang-diagnostic-strict-prototypes, hicpp-uppercase-literal-suffix, cppcoreguidelines-*, performance-*)

/* Zählt das Vorkommen einer Zeichenfolge innerhalb eines Texts */
unsigned long BrbStringCountText(plcstring* pText, plcstring* pFind, unsigned long nTextLen)
{
	UDINT nResult = 0;
	// Wenn die Länge bekannt ist, kann sie übergeben werden
	// Damit entfällt das Aufrufen von strlen, welches bei langen Texten Zeit braucht
	UDINT nLenText = nTextLen;
	if(nTextLen == 0)
	{
		nLenText = strlen(pText);
	}
	UDINT nLenFind = strlen(pFind);
	UDINT nCharIndex = 0;
	// Text von vorne nach hinten durchsuchen
	for(nCharIndex=0; nCharIndex<nLenText; nCharIndex++)
	{
		// Textstelle vergleichen
		if(memcmp((pText + nCharIndex), pFind, nLenFind) == 0)
		{
			// Text gefunden
			nResult += 1;
			nCharIndex += nLenFind-1;
		}
	}
	return nResult;
}

// NOLINTEND(readability-*, bugprone-easily-swappable-parameters, clang-diagnostic-invalid-utf8, clang-diagnostic-invalid-source-encoding, clang-diagnostic-pointer-arith, clang-diagnostic-strict-prototypes, hicpp-uppercase-literal-suffix, cppcoreguidelines-*, performance-*)
```

#### BrbStringRepeat.c - Wiederholt eine Zeichenfolge
```c
#include <bur/plctypes.h>
#ifdef __cplusplus
	extern "C"
	{
#endif

#include "BrbLib.h"
#include <string.h>

#ifdef __cplusplus
	};
#endif

// NOLINTBEGIN(readability-*, bugprone-easily-swappable-parameters, clang-diagnostic-invalid-utf8, clang-diagnostic-invalid-source-encoding, clang-diagnostic-pointer-arith, clang-diagnostic-strict-prototypes, hicpp-uppercase-literal-suffix, cppcoreguidelines-*, performance-*)

/* Wiederholt eine Zeichenfolge bis zu einer angegebenen Zeichenanzahl */
unsigned long BrbStringRepeat(plcstring* pText, unsigned long nTextSize, plcstring* pRepeat, unsigned long nLen)
{
	UDINT nCharCount = 0;
	UDINT nTextOffset = strlen(pText);
	UDINT nRepeatLen = strlen(pRepeat);
	// Länge limitieren
	if(nLen >= nTextSize)
	{
		nLen = nTextSize-1;
	}
	// Gesamten Wiederholtext wiederholend anhängen
	while(nTextOffset+nRepeatLen <= nLen)
	{
		BrbStringAppend(pText, pRepeat, &nTextOffset);
		nCharCount += nRepeatLen;
	}
	// Restliche Zeichen auffüllen
	DINT nCharCountLeft = (DINT)nLen - (DINT)nTextOffset;
	if(nCharCountLeft > 0)
	{
		UDINT nRepeatCharIndex = 0;
		for(nRepeatCharIndex=0; nRepeatCharIndex<(UDINT)nCharCountLeft; nRepeatCharIndex++)
		{
			*(pText + nTextOffset) = *(pRepeat + nRepeatCharIndex);
			nTextOffset++;
			nCharCount++;
		}
		*(pText + nTextOffset) = 0; // String-Abschluss
	}
	return nCharCount;
}

// NOLINTEND(readability-*, bugprone-easily-swappable-parameters, clang-diagnostic-invalid-utf8, clang-diagnostic-invalid-source-encoding, clang-diagnostic-pointer-arith, clang-diagnostic-strict-prototypes, hicpp-uppercase-literal-suffix, cppcoreguidelines-*, performance-*)
```

#### BrbStringCopy.c - Sicheres Kopieren eines Strings
```c
#include <bur/plctypes.h>
#ifdef __cplusplus
	extern "C"
	{
#endif

#include "BrbLib.h"
#include <string.h>

#ifdef __cplusplus
	};
#endif

// NOLINTBEGIN(readability-*, bugprone-easily-swappable-parameters, clang-diagnostic-invalid-utf8, clang-diagnostic-invalid-source-encoding, clang-diagnostic-pointer-arith, clang-diagnostic-strict-prototypes, hicpp-uppercase-literal-suffix, cppcoreguidelines-*, performance-*)

/* Sicheres Kopieren eines Strings */
unsigned long BrbStringCopy(plcstring* pDest, plcstring* pSrc, unsigned long nDestSize)
{
	UDINT nTotalLen = 0;
	if(pDest != 0 && pSrc != 0 && nDestSize > 0)
	{
		// Quellstring kopieren
		UDINT nCopyLen = nTotalLen = strlen(pSrc);
		UDINT nDestLen = nDestSize-1;
		if(nCopyLen > nDestLen)
		{
			nCopyLen = nDestLen;
		}
		memcpy(pDest, pSrc, nCopyLen);
		// Zielstring mit 0 auffüllen (gleichzeitig wird auf jeden Fall der Null-Terminator gesetzt)
		memset((USINT*)pDest+nCopyLen, 0, nDestSize-nCopyLen);
	}
	return nTotalLen;
}

// NOLINTEND(readability-*, bugprone-easily-swappable-parameters, clang-diagnostic-invalid-utf8, clang-diagnostic-invalid-source-encoding, clang-diagnostic-pointer-arith, clang-diagnostic-strict-prototypes, hicpp-uppercase-literal-suffix, cppcoreguidelines-*, performance-*)
```

#### BrbStringCat.c - Sicheres Anfügen eines Strings
```c
#include <bur/plctypes.h>
#ifdef __cplusplus
	extern "C"
	{
#endif

#include "BrbLib.h"
#include <string.h>

#ifdef __cplusplus
	};
#endif

// NOLINTBEGIN(readability-*, bugprone-easily-swappable-parameters, clang-diagnostic-invalid-utf8, clang-diagnostic-invalid-source-encoding, clang-diagnostic-pointer-arith, clang-diagnostic-strict-prototypes, hicpp-uppercase-literal-suffix, cppcoreguidelines-*, performance-*)

/* Sicheres Anhängen an einen String */
unsigned long BrbStringCat(plcstring* pDest, plcstring* pSrc, unsigned long nDestSize)
{
	UDINT nTotalLen = 0;
	if(pDest != 0 && pSrc != 0 && nDestSize > 0)
	{
		// Quellstring anhängen
		UDINT nDestLen = strlen(pDest);
		UDINT nSrcLen = strlen(pSrc);
		nTotalLen = nDestLen + nSrcLen;
		UDINT nSrcLenMax = nDestSize-nDestLen-1;
		if(nSrcLen > nSrcLenMax)
		{
			nSrcLen = nSrcLenMax;
		}
		memcpy(pDest+nDestLen, pSrc, nSrcLen);
		// Zielstring mit 0 auffüllen (gleichzeitig wird auf jeden Fall der Null-Terminator gesetzt)
		memset((USINT*)pDest+nDestLen+nSrcLen, 0, nDestSize-nDestLen-nSrcLen);
	}
	return nTotalLen;
}

// NOLINTEND(readability-*, bugprone-easily-swappable-parameters, clang-diagnostic-invalid-utf8, clang-diagnostic-invalid-source-encoding, clang-diagnostic-pointer-arith, clang-diagnostic-strict-prototypes, hicpp-uppercase-literal-suffix, cppcoreguidelines-*, performance-*)
```

#### Package Logical/Libraries/BrbLib/WcStrings - Unicode-String-Funktionen

#### BrbWcCopyStringToWString.c - Kopiert einen STRING auf einen WSTRING
```c
/********************************************************************
 * COPYRIGHT -- Bernecker + Rainer
 ********************************************************************
 * Library: BrbLib
 * File: BrbWcCopyStringToWString.c
 * Author: niedermeierr
 * Created: April 30, 2016
 ********************************************************************
 * Implementation of library BrbLib
 ********************************************************************/

#include <bur/plctypes.h>
#ifdef __cplusplus
	extern "C"
	{
#endif

#include "BrbLib.h"
#include <string.h>

#ifdef __cplusplus
	};
#endif

// NOLINTBEGIN(readability-*, bugprone-easily-swappable-parameters, clang-diagnostic-invalid-utf8, clang-diagnostic-invalid-source-encoding, clang-diagnostic-pointer-arith, clang-diagnostic-strict-prototypes, hicpp-uppercase-literal-suffix, cppcoreguidelines-*, performance-*)

/* Kopiert einen STRING auf einen WSTRING */
unsigned short BrbWcCopyStringToWString(plcwstring* pWcString, plcstring* pString)
{
	brwcsconv((USINT*)pWcString, (USINT*)pString, brwU8toUC);
	return eBRB_ERR_OK;
}

// NOLINTEND(readability-*, bugprone-easily-swappable-parameters, clang-diagnostic-invalid-utf8, clang-diagnostic-invalid-source-encoding, clang-diagnostic-pointer-arith, clang-diagnostic-strict-prototypes, hicpp-uppercase-literal-suffix, cppcoreguidelines-*, performance-*)
```

#### BrbWcCopyWStringToString.c - Kopiert einen STRING auf einen WSTRING
```c
/********************************************************************
 * COPYRIGHT -- Bernecker + Rainer
 ********************************************************************
 * Library: BrbLib
 * File: BrbWcCopyWStringToString.c
 * Author: niedermeierr
 * Created: Septemer 13, 2021
 ********************************************************************
 * Implementation of library BrbLib
 ********************************************************************/

#include <bur/plctypes.h>
#ifdef __cplusplus
	extern "C"
	{
#endif

#include "BrbLib.h"
#include <string.h>

#ifdef __cplusplus
	};
#endif

// NOLINTBEGIN(readability-*, bugprone-easily-swappable-parameters, clang-diagnostic-invalid-utf8, clang-diagnostic-invalid-source-encoding, clang-diagnostic-pointer-arith, clang-diagnostic-strict-prototypes, hicpp-uppercase-literal-suffix, cppcoreguidelines-*, performance-*)

/* Kopiert einen WSTRING auf einen STRING */
unsigned short BrbWcCopyWStringToString(plcstring* pString, plcwstring* pWcString)
{
	brwcsconv((USINT*)pString, (USINT*)pWcString, brwUCtoU8);
	return eBRB_ERR_OK;
}

// NOLINTEND(readability-*, bugprone-easily-swappable-parameters, clang-diagnostic-invalid-utf8, clang-diagnostic-invalid-source-encoding, clang-diagnostic-pointer-arith, clang-diagnostic-strict-prototypes, hicpp-uppercase-literal-suffix, cppcoreguidelines-*, performance-*)
```

#### BrbWcStringGetIndexOf.c - Gibt den ersten Index eines zu suchenden Textes zurück
```c
/********************************************************************
 * COPYRIGHT -- Bernecker + Rainer
 ********************************************************************
 * Library: BrbLib
 * File: BrbWcStringGetIndexOf.c
 * Author: niedermeierr
 * Created: April 29, 2016
 ********************************************************************
 * Implementation of library BrbLib
 ********************************************************************/

#include <bur/plctypes.h>
#ifdef __cplusplus
	extern "C"
	{
#endif

#include "BrbLib.h"
#include <string.h>

#ifdef __cplusplus
	};
#endif

// NOLINTBEGIN(readability-*, bugprone-easily-swappable-parameters, clang-diagnostic-invalid-utf8, clang-diagnostic-invalid-source-encoding, clang-diagnostic-pointer-arith, clang-diagnostic-strict-prototypes, hicpp-uppercase-literal-suffix, cppcoreguidelines-*, performance-*)

/* Gibt den ersten Index eines zu suchenden Textes zurück */
signed long BrbWcStringGetIndexOf(plcwstring* pText, plcwstring* pFind, unsigned long nTextLen)
{
	DINT nResult = -1;
	// Wenn die Länge bekannt ist, kann sie übergeben werden
	// Damit entfällt das Aufrufen von strlen, welches bei langen Texten Zeit braucht
	UDINT nLenText = nTextLen;
	if(nTextLen == 0)
	{
		nLenText = brwcslen(pText);
	}
	UDINT nByteLenFind = brwcslen(pFind)*2;
	UDINT nCharIndex = 0;
	// Text von vorne nach hinten durchsuchen
	for(nCharIndex=0; nCharIndex<nLenText; nCharIndex++)
	{
		// Textstelle vergleichen
		if(memcmp((pText + nCharIndex), pFind, nByteLenFind) == 0)
		{
			// Text gefunden
			nResult = (DINT)nCharIndex;
			break;
		}
	}
	return nResult;
}

// NOLINTEND(readability-*, bugprone-easily-swappable-parameters, clang-diagnostic-invalid-utf8, clang-diagnostic-invalid-source-encoding, clang-diagnostic-pointer-arith, clang-diagnostic-strict-prototypes, hicpp-uppercase-literal-suffix, cppcoreguidelines-*, performance-*)
```

#### BrbWcStringGetLastIndexOf.c - Gibt den letzten Index eines zu suchenden Textes zurück
```c
/********************************************************************
 * COPYRIGHT -- Bernecker + Rainer
 ********************************************************************
 * Library: BrbLib
 * File: BrbWcStringGetLastIndexOf.c
 * Author: niedermeierr
 * Created: April 29, 2016
 ********************************************************************
 * Implementation of library BrbLib
 ********************************************************************/

#include <bur/plctypes.h>
#ifdef __cplusplus
	extern "C"
	{
#endif

#include "BrbLib.h"
#include <string.h>

#ifdef __cplusplus
	};
#endif

// NOLINTBEGIN(readability-*, bugprone-easily-swappable-parameters, clang-diagnostic-invalid-utf8, clang-diagnostic-invalid-source-encoding, clang-diagnostic-pointer-arith, clang-diagnostic-strict-prototypes, hicpp-uppercase-literal-suffix, cppcoreguidelines-*, performance-*)

/* Gibt den letzten Index eines zu suchenden Textes zurück */
signed long BrbWcStringGetLastIndexOf(plcwstring* pText, plcwstring* pFind, unsigned long nTextLen)
{
	DINT nResult = -1;
	// Wenn die Länge bekannt ist, kann sie übergeben werden
	// Damit entfällt das Aufrufen von strlen, welches bei langen Texten Zeit braucht
	UDINT nLenText = nTextLen;
	if(nTextLen == 0)
	{
		nLenText = brwcslen(pText);
	}
	UDINT nByteLenFind = brwcslen(pFind) * 2;
	DINT nCharIndex = 0;
	// Text von hinten nach vorne durchsuchen
	for(nCharIndex=(DINT)nLenText-1; nCharIndex>=0; nCharIndex--)
	{
		// Textstelle vergleichen
		if(memcmp((pText + nCharIndex), pFind, nByteLenFind) == 0)
		{
			// Text gefunden
			nResult = (DINT)nCharIndex;
			break;
		}
	}
	return nResult;
}

// NOLINTEND(readability-*, bugprone-easily-swappable-parameters, clang-diagnostic-invalid-utf8, clang-diagnostic-invalid-source-encoding, clang-diagnostic-pointer-arith, clang-diagnostic-strict-prototypes, hicpp-uppercase-literal-suffix, cppcoreguidelines-*, performance-*)
```

#### BrbWcStringGetAdrOf.c - Gibt die erste Adresse eines zu suchenden Textes zurück
```c
/********************************************************************
 * COPYRIGHT -- Bernecker + Rainer
 ********************************************************************
 * Library: BrbLib
 * File: BrbWcStringGetAdrOf.c
 * Author: niedermeierr
 * Created: May 02, 2016
 ********************************************************************
 * Implementation of library BrbLib
 ********************************************************************/

#include <bur/plctypes.h>
#ifdef __cplusplus
	extern "C"
	{
#endif

#include "BrbLib.h"
#include <string.h>

#ifdef __cplusplus
	};
#endif

// NOLINTBEGIN(readability-*, bugprone-easily-swappable-parameters, clang-diagnostic-invalid-utf8, clang-diagnostic-invalid-source-encoding, clang-diagnostic-pointer-arith, clang-diagnostic-strict-prototypes, hicpp-uppercase-literal-suffix, cppcoreguidelines-*, performance-*)

/* Gibt die erste Adresse eines zu suchenden Textes zurück */
unsigned long BrbWcStringGetAdrOf(plcwstring* pText, plcwstring* pFind, unsigned long nTextLen)
{
	UDINT nResult = 0;
	// Wenn die Länge bekannt ist, kann sie übergeben werden
	// Damit entfällt das Aufrufen von strlen, welches bei langen Texten Zeit braucht
	UDINT nLenText = nTextLen;
	if(nTextLen == 0)
	{
		nLenText = brwcslen(pText);
	}
	UDINT nByteLenFind = brwcslen(pFind) * 2;
	UDINT nCharIndex = 0;
	// Text von vorne nach hinten durchsuchen
	for(nCharIndex=0; nCharIndex<nLenText; nCharIndex++)
	{
		// Textstelle vergleichen
		if(memcmp((pText + nCharIndex), pFind, nByteLenFind) == 0)
		{
			// Text gefunden
			nResult = (UDINT)(pText + nCharIndex);
			break;
		}
	}
	return nResult;
}

// NOLINTEND(readability-*, bugprone-easily-swappable-parameters, clang-diagnostic-invalid-utf8, clang-diagnostic-invalid-source-encoding, clang-diagnostic-pointer-arith, clang-diagnostic-strict-prototypes, hicpp-uppercase-literal-suffix, cppcoreguidelines-*, performance-*)
```

#### BrbWcStringGetLastAdrOf.c - Gibt die letzte Adresse eines zu suchenden Textes zurück
```c
/********************************************************************
 * COPYRIGHT -- Bernecker + Rainer
 ********************************************************************
 * Library: BrbLib
 * File: BrbWcStringGetLastAdrOf.c
 * Author: niedermeierr
 * Created: May 02, 2016
 ********************************************************************
 * Implementation of library BrbLib
 ********************************************************************/

#include <bur/plctypes.h>
#ifdef __cplusplus
	extern "C"
	{
#endif

#include "BrbLib.h"
#include <string.h>

#ifdef __cplusplus
	};
#endif

// NOLINTBEGIN(readability-*, bugprone-easily-swappable-parameters, clang-diagnostic-invalid-utf8, clang-diagnostic-invalid-source-encoding, clang-diagnostic-pointer-arith, clang-diagnostic-strict-prototypes, hicpp-uppercase-literal-suffix, cppcoreguidelines-*, performance-*)

/* Gibt die letzte Adresse eines zu suchenden Textes zurück */
unsigned long BrbWcStringGetLastAdrOf(plcwstring* pText, plcwstring* pFind, unsigned long nTextLen)
{
	UDINT nResult = 0;
	// Wenn die Länge bekannt ist, kann sie übergeben werden
	// Damit entfällt das Aufrufen von strlen, welches bei langen Texten Zeit braucht
	UDINT nLenText = nTextLen;
	if(nTextLen == 0)
	{
		nLenText = brwcslen(pText);
	}
	UDINT nByteLenFind = brwcslen(pFind) * 2;
	DINT nCharIndex = 0;
	// Text von hinten nach vorne durchsuchen
	for(nCharIndex=(DINT)nLenText-1; nCharIndex>=0; nCharIndex--)
	{
		// Textstelle vergleichen
		if(memcmp((pText + nCharIndex), pFind, nByteLenFind) == 0)
		{
			// Text gefunden
			nResult = (UDINT)(pText + nCharIndex);
			break;
		}
	}
	return nResult;
}

// NOLINTEND(readability-*, bugprone-easily-swappable-parameters, clang-diagnostic-invalid-utf8, clang-diagnostic-invalid-source-encoding, clang-diagnostic-pointer-arith, clang-diagnostic-strict-prototypes, hicpp-uppercase-literal-suffix, cppcoreguidelines-*, performance-*)
```

#### BrbWcStringStartsWith.c - Gibt zurück, ob ein Text mit einer bestimmten Zeichenfolge beginnt
```c
/********************************************************************
 * COPYRIGHT -- Bernecker + Rainer
 ********************************************************************
 * Library: BrbLib
 * File: BrbWcStringStartsWith.c
 * Author: niedermeierr
 * Created: May 02, 2016
 ********************************************************************
 * Implementation of library BrbLib
 ********************************************************************/

#include <bur/plctypes.h>
#ifdef __cplusplus
	extern "C"
	{
#endif

#include "BrbLib.h"
#include <string.h>

#ifdef __cplusplus
	};
#endif

// NOLINTBEGIN(readability-*, bugprone-easily-swappable-parameters, clang-diagnostic-invalid-utf8, clang-diagnostic-invalid-source-encoding, clang-diagnostic-pointer-arith, clang-diagnostic-strict-prototypes, hicpp-uppercase-literal-suffix, cppcoreguidelines-*, performance-*)

/* Gibt zurück, ob ein Text mit einer bestimmten Zeichenfolge beginnt */
plcbit BrbWcStringStartsWith(plcwstring* pText, plcwstring* pFind)
{
	BOOL bResult = 0;
	UDINT nByteLenFind = brwcslen(pFind) * 2;
	if(memcmp(pText, pFind, nByteLenFind) == 0)
	{
		bResult = 1;
	}
	return bResult;
}

// NOLINTEND(readability-*, bugprone-easily-swappable-parameters, clang-diagnostic-invalid-utf8, clang-diagnostic-invalid-source-encoding, clang-diagnostic-pointer-arith, clang-diagnostic-strict-prototypes, hicpp-uppercase-literal-suffix, cppcoreguidelines-*, performance-*)
```

#### BrbWcStringEndsWith.c - Gibt zurück, ob ein Text mit einer bestimmten Zeichenfolge endet
```c
/********************************************************************
 * COPYRIGHT -- Bernecker + Rainer
 ********************************************************************
 * Library: BrbLib
 * File: BrbWcStringEndsWith.c
 * Author: niedermeierr
 * Created: May 02, 2016
 ********************************************************************
 * Implementation of library BrbLib
 ********************************************************************/

#include <bur/plctypes.h>
#ifdef __cplusplus
	extern "C"
	{
#endif

#include "BrbLib.h"
#include <string.h>

#ifdef __cplusplus
	};
#endif

// NOLINTBEGIN(readability-*, bugprone-easily-swappable-parameters, clang-diagnostic-invalid-utf8, clang-diagnostic-invalid-source-encoding, clang-diagnostic-pointer-arith, clang-diagnostic-strict-prototypes, hicpp-uppercase-literal-suffix, cppcoreguidelines-*, performance-*)

/* Gibt zurück, ob ein Text mit einer bestimmten Zeichenfolge endet */
plcbit BrbWcStringEndsWith(plcwstring* pText, plcwstring* pFind)
{
	BOOL bResult = 0;
	UDINT nLenText = brwcslen(pText);
	UDINT nLenFind = brwcslen(pFind);
	UDINT nByteLenFind = nLenFind * 2;
	if(nLenText >= nLenFind)
	{
		if(memcmp(pText + nLenText - nLenFind, pFind, nByteLenFind) == 0)
		{
			bResult = 1;
		}
	}
	return bResult;
}

// NOLINTEND(readability-*, bugprone-easily-swappable-parameters, clang-diagnostic-invalid-utf8, clang-diagnostic-invalid-source-encoding, clang-diagnostic-pointer-arith, clang-diagnostic-strict-prototypes, hicpp-uppercase-literal-suffix, cppcoreguidelines-*, performance-*)
```

#### BrbWcStringGetSubText.c - Gibt eine Zeichenfolge innerhalb eines Textes zurück
```c
/********************************************************************
 * COPYRIGHT -- Bernecker + Rainer
 ********************************************************************
 * Library: BrbLib
 * File: BrbWcStringGetSubText.c
 * Author: niedermeierr
 * Created: May 02, 2016
 ********************************************************************
 * Implementation of library BrbLib
 ********************************************************************/

#include <bur/plctypes.h>
#ifdef __cplusplus
	extern "C"
	{
#endif

#include "BrbLib.h"
#include <string.h>

#ifdef __cplusplus
	};
#endif

// NOLINTBEGIN(readability-*, bugprone-easily-swappable-parameters, clang-diagnostic-invalid-utf8, clang-diagnostic-invalid-source-encoding, clang-diagnostic-pointer-arith, clang-diagnostic-strict-prototypes, hicpp-uppercase-literal-suffix, cppcoreguidelines-*, performance-*)

/* Gibt eine Zeichenfolge innerhalb eines Textes zurück */
unsigned long BrbWcStringGetSubText(plcwstring* pText, unsigned long nIndex, unsigned long nLen, plcwstring* pSubText)
{
	UDINT nByteLen = nLen * 2;
	memcpy(pSubText, (pText + nIndex), nByteLen);
	pSubText[nLen] = 0; // NullTerminierung
	return (UDINT)(pText + nIndex + nLen);
}

// NOLINTEND(readability-*, bugprone-easily-swappable-parameters, clang-diagnostic-invalid-utf8, clang-diagnostic-invalid-source-encoding, clang-diagnostic-pointer-arith, clang-diagnostic-strict-prototypes, hicpp-uppercase-literal-suffix, cppcoreguidelines-*, performance-*)
```

#### BrbWcStringGetSubTextByLen.c - Gibt eine Zeichenfolge innerhalb eines Textes zurück
```c
/********************************************************************
 * COPYRIGHT -- Bernecker + Rainer
 ********************************************************************
 * Library: BrbLib
 * File: BrbWcStringGetSubTextByLen.c
 * Author: niedermeierr
 * Created: May 02, 2016
 ********************************************************************
 * Implementation of library BrbLib
 ********************************************************************/

#include <bur/plctypes.h>
#ifdef __cplusplus
	extern "C"
	{
#endif

#include "BrbLib.h"
#include <string.h>

#ifdef __cplusplus
	};
#endif

// NOLINTBEGIN(readability-*, bugprone-easily-swappable-parameters, clang-diagnostic-invalid-utf8, clang-diagnostic-invalid-source-encoding, clang-diagnostic-pointer-arith, clang-diagnostic-strict-prototypes, hicpp-uppercase-literal-suffix, cppcoreguidelines-*, performance-*)

/* Gibt eine Zeichenfolge innerhalb eines Textes zurück */
unsigned long BrbWcStringGetSubTextByLen(plcwstring* pStart, unsigned long nLen, plcwstring* pSubText)
{
	UDINT nByteLen = nLen * 2;
	memcpy(pSubText, pStart, nByteLen);
	pSubText[nLen] = 0; // NullTerminierung
	return (UDINT)(pStart + nLen);
}

// NOLINTEND(readability-*, bugprone-easily-swappable-parameters, clang-diagnostic-invalid-utf8, clang-diagnostic-invalid-source-encoding, clang-diagnostic-pointer-arith, clang-diagnostic-strict-prototypes, hicpp-uppercase-literal-suffix, cppcoreguidelines-*, performance-*)
```

#### BrbWcStringGetSubTextByAdr.c - Gibt eine Zeichenfolge innerhalb eines Textes zurück
```c
/********************************************************************
 * COPYRIGHT -- Bernecker + Rainer
 ********************************************************************
 * Library: BrbLib
 * File: BrbWcStringGetSubTextByAdr.c
 * Author: niedermeierr
 * Created: May 02, 2016
 ********************************************************************
 * Implementation of library BrbLib
 ********************************************************************/

#include <bur/plctypes.h>
#ifdef __cplusplus
	extern "C"
	{
#endif

#include "BrbLib.h"
#include <string.h>

#ifdef __cplusplus
	};
#endif

// NOLINTBEGIN(readability-*, bugprone-easily-swappable-parameters, clang-diagnostic-invalid-utf8, clang-diagnostic-invalid-source-encoding, clang-diagnostic-pointer-arith, clang-diagnostic-strict-prototypes, hicpp-uppercase-literal-suffix, cppcoreguidelines-*, performance-*)

/* Gibt eine Zeichenfolge innerhalb eines Textes zurück */
unsigned long BrbWcStringGetSubTextByAdr(plcwstring* pStart, plcwstring* pEnd, plcwstring* pSubText)
{
	UDINT nResult = 0;
	if(pEnd > pStart)
	{
		UDINT nLen = (UDINT)(pEnd - pStart);
		nResult = BrbWcStringGetSubTextByLen(pStart, nLen, pSubText);
	}
	return nResult;
}

// NOLINTEND(readability-*, bugprone-easily-swappable-parameters, clang-diagnostic-invalid-utf8, clang-diagnostic-invalid-source-encoding, clang-diagnostic-pointer-arith, clang-diagnostic-strict-prototypes, hicpp-uppercase-literal-suffix, cppcoreguidelines-*, performance-*)
```

#### BrbWcStringAppend.c - Hängt eine Zeichenfolge an einen Text (Ersatz für brwcscat)
```c
/********************************************************************
 * COPYRIGHT -- Bernecker + Rainer
 ********************************************************************
 * Library: BrbLib
 * File: BrbWcStringAppend.c
 * Author: niedermeierr
 * Created: May 02, 2016
 ********************************************************************
 * Implementation of library BrbLib
 ********************************************************************/

#include <bur/plctypes.h>
#ifdef __cplusplus
	extern "C"
	{
#endif

#include "BrbLib.h"
#include <string.h>

#ifdef __cplusplus
	};
#endif

// NOLINTBEGIN(readability-*, bugprone-easily-swappable-parameters, clang-diagnostic-invalid-utf8, clang-diagnostic-invalid-source-encoding, clang-diagnostic-pointer-arith, clang-diagnostic-strict-prototypes, hicpp-uppercase-literal-suffix, cppcoreguidelines-*, performance-*)

/* Hängt eine Zeichenfolge an einen Text (Ersatz für brwcscat) */
unsigned long BrbWcStringAppend(plcwstring* pText, plcwstring* pTextAppend, unsigned long* pTextOffset)
{
	UDINT nAppendLen = brwcslen(pTextAppend);
	UDINT nAppendByteLen = nAppendLen * 2;
	memcpy(pText + *pTextOffset, pTextAppend, nAppendByteLen);
	*pTextOffset += nAppendLen;
	*(pText + *pTextOffset) = 0; // String-Abschluss
	return nAppendLen;
}

// NOLINTEND(readability-*, bugprone-easily-swappable-parameters, clang-diagnostic-invalid-utf8, clang-diagnostic-invalid-source-encoding, clang-diagnostic-pointer-arith, clang-diagnostic-strict-prototypes, hicpp-uppercase-literal-suffix, cppcoreguidelines-*, performance-*)
```

#### BrbWcStringCut.c - Schneidet eine Zeichenfolge aus einem Text heraus
```c
/********************************************************************
 * COPYRIGHT -- Bernecker + Rainer
 ********************************************************************
 * Library: BrbLib
 * File: BrbWcStringCut.c
 * Author: niedermeierr
 * Created: May 02, 2016
 ********************************************************************
 * Implementation of library BrbLib
 ********************************************************************/

#include <bur/plctypes.h>
#ifdef __cplusplus
	extern "C"
	{
#endif

#include "BrbLib.h"
#include <string.h>

#ifdef __cplusplus
	};
#endif

// NOLINTBEGIN(readability-*, bugprone-easily-swappable-parameters, clang-diagnostic-invalid-utf8, clang-diagnostic-invalid-source-encoding, clang-diagnostic-pointer-arith, clang-diagnostic-strict-prototypes, hicpp-uppercase-literal-suffix, cppcoreguidelines-*, performance-*)

/* Schneidet eine Zeichenfolge aus einem Text heraus */
unsigned long BrbWcStringCut(plcwstring* pText, unsigned long nCutIndex, unsigned long nCutLen, plcwstring* pCut)
{
	UDINT nResult = 0;
	UDINT nCutByteLen = nCutLen * 2;
	UDINT nTextLen = brwcslen(pText);
	if(nCutIndex+nCutLen > nTextLen)
	{
		nCutLen = nTextLen-nCutIndex;
	}
	if(pCut != 0)
	{
		// Herauszuschneidenden String kopieren
		memcpy(pCut, (pText + nCutIndex), nCutByteLen);
		*(pCut + nCutLen) = 0;
	}
	UDINT nRestByteLen = (nTextLen - nCutIndex - nCutLen + 1) * 2;
	// Zeichen nach dem Cut nach vorne ziehen
	memmove((pText + nCutIndex), (pText + nCutIndex + nCutLen), nRestByteLen);
	nResult = (UDINT)(pText + nCutIndex + nCutLen);
	return nResult;
}

// NOLINTEND(readability-*, bugprone-easily-swappable-parameters, clang-diagnostic-invalid-utf8, clang-diagnostic-invalid-source-encoding, clang-diagnostic-pointer-arith, clang-diagnostic-strict-prototypes, hicpp-uppercase-literal-suffix, cppcoreguidelines-*, performance-*)
```

#### BrbWcStringInsert.c - Fügt eine Zeichenfolge in einen Text ein
```c
/********************************************************************
 * COPYRIGHT -- Bernecker + Rainer
 ********************************************************************
 * Library: BrbLib
 * File: BrbWcStringInsert.c
 * Author: niedermeierr
 * Created: May 02, 2016
 ********************************************************************
 * Implementation of library BrbLib
 ********************************************************************/

#include <bur/plctypes.h>
#ifdef __cplusplus
	extern "C"
	{
#endif

#include "BrbLib.h"
#include <string.h>

#ifdef __cplusplus
	};
#endif

// NOLINTBEGIN(readability-*, bugprone-easily-swappable-parameters, clang-diagnostic-invalid-utf8, clang-diagnostic-invalid-source-encoding, clang-diagnostic-pointer-arith, clang-diagnostic-strict-prototypes, hicpp-uppercase-literal-suffix, cppcoreguidelines-*, performance-*)

/* Fügt eine Zeichenfolge in einen Text ein */
unsigned long BrbWcStringInsert(plcwstring* pText, unsigned long nInsertIndex, plcwstring* pInsert)
{
	UDINT nResult = 0;
	UDINT nTextLen = brwcslen(pText);
	UDINT nInsertLen = brwcslen(pInsert);
	UDINT nInsertByteLen = nInsertLen * 2;
	UDINT nRestByteLen = (nTextLen - nInsertIndex + 1) * 2;
	// Zeichen am Index nach hinten schieben
	memmove((pText + nInsertIndex + nInsertLen), (pText + nInsertIndex), nRestByteLen);
	memcpy((pText + nInsertIndex), pInsert, nInsertByteLen);
	nResult = (UDINT)(pText + nInsertIndex + nInsertLen);
	return nResult;
}

// NOLINTEND(readability-*, bugprone-easily-swappable-parameters, clang-diagnostic-invalid-utf8, clang-diagnostic-invalid-source-encoding, clang-diagnostic-pointer-arith, clang-diagnostic-strict-prototypes, hicpp-uppercase-literal-suffix, cppcoreguidelines-*, performance-*)
```

#### BrbWcStringReplace.c - Ersetzt eine Zeichenfolge in einem Text durch eine andere
```c
/********************************************************************
 * COPYRIGHT -- Bernecker + Rainer
 ********************************************************************
 * Library: BrbLib
 * File: BrbWcStringReplace.c
 * Author: niedermeierr
 * Created: May 02, 2016
 ********************************************************************
 * Implementation of library BrbLib
 ********************************************************************/

#include <bur/plctypes.h>
#ifdef __cplusplus
	extern "C"
	{
#endif

#include "BrbLib.h"
#include <string.h>

#ifdef __cplusplus
	};
#endif

// NOLINTBEGIN(readability-*, bugprone-easily-swappable-parameters, clang-diagnostic-invalid-utf8, clang-diagnostic-invalid-source-encoding, clang-diagnostic-pointer-arith, clang-diagnostic-strict-prototypes, hicpp-uppercase-literal-suffix, cppcoreguidelines-*, performance-*)

/* Ersetzt eine Zeichenfolge in einem Text durch eine andere */
unsigned long BrbWcStringReplace(plcwstring* pText, plcwstring* pFind, plcwstring* pReplace)
{
	UDINT nResult = 0;
	UDINT nTextLen = brwcslen(pText);
	UDINT nFindLen = brwcslen(pFind);
	UDINT nFindByteLen = nFindLen * 2;
	UDINT nReplaceLen = brwcslen(pReplace);
	UDINT nReplaceByteLen = nReplaceLen * 2;
	DINT nDiff = (DINT)nReplaceLen - (DINT)nFindLen;
	UDINT nCharIndex = 0;
	// Text von vorne nach hinten durchsuchen
	while(1==1)
	{
		// Textstelle vergleichen
		if(memcmp((pText + nCharIndex), pFind, nFindByteLen) == 0)
		{
			// Text gefunden
			if(nDiff > 0)
			{
				// Replace ist länger
				UDINT nRestByteLen = (nTextLen - nCharIndex + 1) * 2;
				memmove((pText + nCharIndex + nDiff), (pText + nCharIndex), nRestByteLen);
				memcpy((pText + nCharIndex), pReplace, nReplaceByteLen);
				nTextLen += (UDINT)nDiff;
				nCharIndex += nReplaceLen;
				nResult += 1;
			}
			else if(nDiff < 0)
			{
				// Replace ist kürzer
				UDINT nRestByteLen = (UDINT)((DINT)nTextLen - (DINT)nCharIndex + nDiff + 1) * 2;
				memmove((pText + nCharIndex), (pText + nCharIndex - nDiff), nRestByteLen);
				memcpy((pText + nCharIndex), pReplace, nReplaceByteLen);
				nTextLen = (UDINT)((DINT)nTextLen + nDiff);
				nCharIndex += nReplaceLen;
				nResult += 1;
			}
			else
			{
				// Zeichenfolgen sind gleich lang
				memcpy((pText + nCharIndex), pReplace, nReplaceByteLen);
				nCharIndex += nReplaceLen;
				nResult += 1;
			}
		}
		else
		{
			nCharIndex += 1;
		}
		if(nCharIndex>=nTextLen)
		{
			break;
		}
	}
	return nResult;
}

// NOLINTEND(readability-*, bugprone-easily-swappable-parameters, clang-diagnostic-invalid-utf8, clang-diagnostic-invalid-source-encoding, clang-diagnostic-pointer-arith, clang-diagnostic-strict-prototypes, hicpp-uppercase-literal-suffix, cppcoreguidelines-*, performance-*)
```

#### BrbWcStringPadLeft.c - Füllt einen String auf der linken Seite mit einem Füllzeichen auf eine bestimme Länge
```c
/********************************************************************
 * COPYRIGHT -- Bernecker + Rainer
 ********************************************************************
 * Library: BrbLib
 * File: BrbWcStringPadLeft.c
 * Author: niedermeierr
 * Created: May 03, 2016
 ********************************************************************
 * Implementation of library BrbLib
 ********************************************************************/

#include <bur/plctypes.h>
#ifdef __cplusplus
	extern "C"
	{
#endif

#include "BrbLib.h"
#include <string.h>

#ifdef __cplusplus
	};
#endif

// NOLINTBEGIN(readability-*, bugprone-easily-swappable-parameters, clang-diagnostic-invalid-utf8, clang-diagnostic-invalid-source-encoding, clang-diagnostic-pointer-arith, clang-diagnostic-strict-prototypes, hicpp-uppercase-literal-suffix, cppcoreguidelines-*, performance-*)

/* Füllt einen String auf der linken Seite mit einem Füllzeichen auf eine bestimme Länge */
plcbit BrbWcStringPadLeft(plcwstring* pText, plcwstring* pFillChar, unsigned long nLen)
{
	BOOL bResult = 0;
	UDINT nTextLen = brwcslen(pText);
	UDINT nTextByteLen = nTextLen * 2;
	DINT nFillLen = (DINT)nLen - (DINT)nTextLen;
	UINT* pChar = (UINT*)pText;
	if(nFillLen > 0)
	{
		// Text nach rechts schieben
		memmove(pText+nFillLen, pText, nTextByteLen+2);
		// Füllzeichen einsetzen
		while(pChar < (UINT*)(pText+nFillLen))
		{
			*pChar = *pFillChar;
			pChar++;
		}
		bResult = 1;
	}
	return bResult;
}

// NOLINTEND(readability-*, bugprone-easily-swappable-parameters, clang-diagnostic-invalid-utf8, clang-diagnostic-invalid-source-encoding, clang-diagnostic-pointer-arith, clang-diagnostic-strict-prototypes, hicpp-uppercase-literal-suffix, cppcoreguidelines-*, performance-*)
```

#### BrbWcStringPadRight.c - Füllt einen String auf der rechten Seite mit einem Füllzeichen auf eine bestimme Länge
```c
/********************************************************************
 * COPYRIGHT -- Bernecker + Rainer
 ********************************************************************
 * Library: BrbLib
 * File: BrbWcStringPadRight.c
 * Author: niedermeierr
 * Created: May 03, 2016
 ********************************************************************
 * Implementation of library BrbLib
 ********************************************************************/

#include <bur/plctypes.h>
#ifdef __cplusplus
	extern "C"
	{
#endif

#include "BrbLib.h"
#include <string.h>

#ifdef __cplusplus
	};
#endif

// NOLINTBEGIN(readability-*, bugprone-easily-swappable-parameters, clang-diagnostic-invalid-utf8, clang-diagnostic-invalid-source-encoding, clang-diagnostic-pointer-arith, clang-diagnostic-strict-prototypes, hicpp-uppercase-literal-suffix, cppcoreguidelines-*, performance-*)

/* Füllt einen String auf der rechten Seite mit einem Füllzeichen auf eine bestimme Länge */
plcbit BrbWcStringPadRight(plcwstring* pText, plcwstring* pFillChar, unsigned long nLen)
{
	BOOL bResult = 0;
	UDINT nTextLen = brwcslen(pText);
	DINT nFillLen = (DINT)nLen - (DINT)nTextLen;
	UINT* pChar = (UINT*)pText + nTextLen;
	if(nFillLen > 0)
	{
		// Füllzeichen einsetzen
		while(pChar < (UINT*)(pText+nLen))
		{
			*pChar = *pFillChar;
			pChar++;
		}
		bResult = 1;
	}
	// Terminierung
	*pChar = 0;
	return bResult;
}

// NOLINTEND(readability-*, bugprone-easily-swappable-parameters, clang-diagnostic-invalid-utf8, clang-diagnostic-invalid-source-encoding, clang-diagnostic-pointer-arith, clang-diagnostic-strict-prototypes, hicpp-uppercase-literal-suffix, cppcoreguidelines-*, performance-*)
```

#### BrbWcStringTrimLeft.c - Schneidet eine Zeichenfolge auf der linken Seite eines Textes heraus
```c
/********************************************************************
 * COPYRIGHT -- Bernecker + Rainer
 ********************************************************************
 * Library: BrbLib
 * File: BrbWcStringTrimLeft.c
 * Author: niedermeierr
 * Created: May 03, 2016
 ********************************************************************
 * Implementation of library BrbLib
 ********************************************************************/

#include <bur/plctypes.h>
#ifdef __cplusplus
	extern "C"
	{
#endif

#include "BrbLib.h"
#include <string.h>

#ifdef __cplusplus
	};
#endif

// NOLINTBEGIN(readability-*, bugprone-easily-swappable-parameters, clang-diagnostic-invalid-utf8, clang-diagnostic-invalid-source-encoding, clang-diagnostic-pointer-arith, clang-diagnostic-strict-prototypes, hicpp-uppercase-literal-suffix, cppcoreguidelines-*, performance-*)

/* Schneidet eine Zeichenfolge auf der linken Seite eines Textes heraus */
plcbit BrbWcStringTrimLeft(plcwstring* pText, plcwstring* pTrim)
{
	BOOL bResult = 0;
	UDINT nTrimLen = brwcslen(pTrim);
	BOOL bLeave = 0;
	do
	{
		if(BrbWcStringStartsWith(pText, pTrim) == 1)
		{
			BrbWcStringCut(pText, 0, nTrimLen, 0);
			bResult = 1;
		}
		else
		{
			bLeave = 1;
		}
	} while(bLeave == 0);
	return bResult;
}

// NOLINTEND(readability-*, bugprone-easily-swappable-parameters, clang-diagnostic-invalid-utf8, clang-diagnostic-invalid-source-encoding, clang-diagnostic-pointer-arith, clang-diagnostic-strict-prototypes, hicpp-uppercase-literal-suffix, cppcoreguidelines-*, performance-*)
```

#### BrbWcStringTrimRight.c - Schneidet eine Zeichenfolge auf der rechten Seite eines Textes heraus
```c
/********************************************************************
 * COPYRIGHT -- Bernecker + Rainer
 ********************************************************************
 * Library: BrbLib
 * File: BrbWcStringTrimRight.c
 * Author: niedermeierr
 * Created: May 04, 2016
 ********************************************************************
 * Implementation of library BrbLib
 ********************************************************************/

#include <bur/plctypes.h>
#ifdef __cplusplus
	extern "C"
	{
#endif

#include "BrbLib.h"
#include <string.h>

#ifdef __cplusplus
	};
#endif

// NOLINTBEGIN(readability-*, bugprone-easily-swappable-parameters, clang-diagnostic-invalid-utf8, clang-diagnostic-invalid-source-encoding, clang-diagnostic-pointer-arith, clang-diagnostic-strict-prototypes, hicpp-uppercase-literal-suffix, cppcoreguidelines-*, performance-*)

/* Schneidet eine Zeichenfolge auf der rechten Seite eines Textes heraus */
plcbit BrbWcStringTrimRight(plcwstring* pText, plcwstring* pTrim)
{
	BOOL bResult = 0;
	UDINT nTrimLen = brwcslen(pTrim);
	BOOL bLeave = 0;
	do
	{
		if(BrbWcStringEndsWith(pText, pTrim) == 1)
		{
			UDINT nTextLen = brwcslen(pText);
			BrbWcStringCut(pText, nTextLen-nTrimLen, nTrimLen, 0);
			bResult = 1;
		}
		else
		{
			bLeave = 1;
		}
	} while(bLeave == 0);
	return bResult;
}

// NOLINTEND(readability-*, bugprone-easily-swappable-parameters, clang-diagnostic-invalid-utf8, clang-diagnostic-invalid-source-encoding, clang-diagnostic-pointer-arith, clang-diagnostic-strict-prototypes, hicpp-uppercase-literal-suffix, cppcoreguidelines-*, performance-*)
```

#### BrbWcStringToUpper.c - Konvertiert einen String zu Großbuchstaben
```c
/********************************************************************
 * COPYRIGHT -- Bernecker + Rainer
 ********************************************************************
 * Library: BrbLib
 * File: BrbWcStringToUpper.c
 * Author: niedermeierr
 * Created: May 04, 2016
 ********************************************************************
 * Implementation of library BrbLib
 ********************************************************************/

#include <bur/plctypes.h>
#ifdef __cplusplus
	extern "C"
	{
#endif

#include "BrbLib.h"
#include <string.h>

#ifdef __cplusplus
	};
#endif

// NOLINTBEGIN(readability-*, bugprone-easily-swappable-parameters, clang-diagnostic-invalid-utf8, clang-diagnostic-invalid-source-encoding, clang-diagnostic-pointer-arith, clang-diagnostic-strict-prototypes, hicpp-uppercase-literal-suffix, cppcoreguidelines-*, performance-*)

/* Konvertiert einen WcString zu Großbuchstaben */
plcbit BrbWcStringToUpper(plcwstring* pText)
{
	BOOL bResult = 0;
	UDINT nTextLen = brwcslen(pText);
	UDINT nIndex = 0;
	UINT* pChar = 0;
	for(nIndex=0; nIndex<nTextLen; nIndex++)
	{
		pChar = (UINT*)(pText + nIndex);
		if(*pChar >= 97 && *pChar <= 122)
		{
			*pChar = *pChar - 32;
			bResult = 1;
		}
	}
	return bResult;
}

// NOLINTEND(readability-*, bugprone-easily-swappable-parameters, clang-diagnostic-invalid-utf8, clang-diagnostic-invalid-source-encoding, clang-diagnostic-pointer-arith, clang-diagnostic-strict-prototypes, hicpp-uppercase-literal-suffix, cppcoreguidelines-*, performance-*)
```

#### BrbWcStringToLower.c - Konvertiert einen WcString zu Kleinbuchstaben
```c
/********************************************************************
 * COPYRIGHT -- Bernecker + Rainer
 ********************************************************************
 * Library: BrbLib
 * File: BrbWcStringToLower.c
 * Author: niedermeierr
 * Created: May 04, 2016
 ********************************************************************
 * Implementation of library BrbLib
 ********************************************************************/

#include <bur/plctypes.h>
#ifdef __cplusplus
	extern "C"
	{
#endif

#include "BrbLib.h"
#include <string.h>

#ifdef __cplusplus
	};
#endif

// NOLINTBEGIN(readability-*, bugprone-easily-swappable-parameters, clang-diagnostic-invalid-utf8, clang-diagnostic-invalid-source-encoding, clang-diagnostic-pointer-arith, clang-diagnostic-strict-prototypes, hicpp-uppercase-literal-suffix, cppcoreguidelines-*, performance-*)

/* Konvertiert einen WcString zu Kleinbuchstaben */
plcbit BrbWcStringToLower(plcwstring* pText)
{
	BOOL bResult = 0;
	UDINT nTextLen = brwcslen(pText);
	UDINT nIndex = 0;
	UINT* pChar = 0;
	for(nIndex=0; nIndex<nTextLen; nIndex++)
	{
		pChar = (UINT*)(pText + nIndex);
		if(*pChar >= 65 && *pChar <= 90)
		{
			*pChar = *pChar + 32;
			bResult = 1;
		}
	}
	return bResult;
}

// NOLINTEND(readability-*, bugprone-easily-swappable-parameters, clang-diagnostic-invalid-utf8, clang-diagnostic-invalid-source-encoding, clang-diagnostic-pointer-arith, clang-diagnostic-strict-prototypes, hicpp-uppercase-literal-suffix, cppcoreguidelines-*, performance-*)
```

#### BrbWcStringIsNumerical.c - Gibt zurück, ob ein Text eine Nummer enthält
```c
/********************************************************************
 * COPYRIGHT -- Bernecker + Rainer
 ********************************************************************
 * Library: BrbLib
 * File: BrbWcStringIsNumerical.c
 * Author: niedermeierr
 * Created: May 04, 2016
 ********************************************************************
 * Implementation of library BrbLib
 ********************************************************************/

#include <bur/plctypes.h>
#ifdef __cplusplus
	extern "C"
	{
#endif

#include "BrbLib.h"
#include <string.h>

#ifdef __cplusplus
	};
#endif

// NOLINTBEGIN(readability-*, bugprone-easily-swappable-parameters, clang-diagnostic-invalid-utf8, clang-diagnostic-invalid-source-encoding, clang-diagnostic-pointer-arith, clang-diagnostic-strict-prototypes, hicpp-uppercase-literal-suffix, cppcoreguidelines-*, performance-*)

/* Gibt zurück, ob ein Text eine Nummer enthält */
plcbit BrbWcStringIsNumerical(plcwstring* pText) // NOLINT(readability-function-cognitive-complexity)
{
	BOOL bResult = 1;
	UDINT nTextLen = brwcslen(pText);
	if(nTextLen == 0)
	{
		bResult = 0;
	}
	else
	{
		UDINT nIndex = 0;
		UINT* pChar = 0;
		UINT nCountSeparator = 0;
		DINT nIndexExp = -1;
		for(nIndex=0; nIndex<nTextLen; nIndex++)
		{
			pChar = (UINT*)(pText + nIndex);
			// NOLINTBEGIN(bugprone-branch-clone)
			if(*pChar == 43)
			{
				// Plus
				if(nIndex != 0 && nIndexExp != (DINT)nIndex-1)
				{
					// Nicht am Anfang oder nach "e"
					bResult = 0;
					break;
				}
			}
			else if(*pChar == 45)
			{
				// Minus
				if(nIndex != 0 && nIndexExp != (DINT)nIndex-1)
				{
					// Nicht am Anfang oder nach "e"
					bResult = 0;
					break;
				}
			}
			else if(*pChar == 44)
			{
				// Komma
				nCountSeparator++;
				if(nCountSeparator > 1)
				{
					// Mehr als 1 Separartor
					bResult = 0;
					break;
				}
			}
			else if(*pChar == 46)
			{
				// Punkt
				nCountSeparator++;
				if(nCountSeparator > 1)
				{
					// Mehr als 1 Separartor
					bResult = 0;
					break;
				}
			}
			else if(*pChar == 101)
			{
				// e
				if(nIndexExp == -1)
				{
					nIndexExp = (DINT)nIndex;
					if(nIndex >= nTextLen-1)
					{
						// Nach "e" folgt nichts
						bResult = 0;
						break;
					}
				}
				else
				{
					// Zweites "e"
					bResult = 0;
					break;
				}
			}
			else if(!(*pChar >= 48 && *pChar <= 57))
			{
				bResult = 0;
				break;
			}
			// NOLINTEND(bugprone-branch-clone)
		}
	}
	return bResult;
}

// NOLINTEND(readability-*, bugprone-easily-swappable-parameters, clang-diagnostic-invalid-utf8, clang-diagnostic-invalid-source-encoding, clang-diagnostic-pointer-arith, clang-diagnostic-strict-prototypes, hicpp-uppercase-literal-suffix, cppcoreguidelines-*, performance-*)
```

#### BrbWcStringIsHex.c - Gibt zurück, ob ein Text eine hexadezimale Nummer enthält
```c
/********************************************************************
 * COPYRIGHT -- Bernecker + Rainer
 ********************************************************************
 * Library: BrbLib
 * File: BrbWcStringIsHex.c
 * Author: niedermeierr
 * Created: January 17, 2017
 ********************************************************************
 * Implementation of library BrbLib
 ********************************************************************/

#include <bur/plctypes.h>
#ifdef __cplusplus
	extern "C"
	{
#endif

	#include "BrbLib.h"

#ifdef __cplusplus
	};
#endif

// NOLINTBEGIN(readability-*, bugprone-easily-swappable-parameters, clang-diagnostic-invalid-utf8, clang-diagnostic-invalid-source-encoding, clang-diagnostic-pointer-arith, clang-diagnostic-strict-prototypes, hicpp-uppercase-literal-suffix, cppcoreguidelines-*, performance-*)

/* Gibt zurück, ob ein Text eine hexadezimale Nummer enthält */
plcbit BrbWcStringIsHex(plcwstring* pText, plcbit bLowCaseAllowed)
{
	BOOL bResult = 1;
	UDINT nTextLen = brwcslen(pText);
	if(nTextLen == 0)
	{
		bResult = 0;
	}
	else
	{
		UDINT nIndex = 0;
		UINT* pChar = 0;
		for(nIndex=0; nIndex<nTextLen; nIndex++)
		{
			pChar = (UINT*)(pText + nIndex);
			// NOLINTBEGIN(bugprone-branch-clone)
			if((*pChar >= 48 && *pChar <= 57)) // 0..9
			{
			}
			else if((*pChar >= 65 && *pChar <= 70)) // A..F
			{
			}
			else if((*pChar >= 97 && *pChar <= 102) && bLowCaseAllowed == 1) // a..f
			{
			}
			else
			{
				bResult = 0;
				break;
			}
			// NOLINTEND(bugprone-branch-clone)
		}
	}
	return bResult;
}

// NOLINTEND(readability-*, bugprone-easily-swappable-parameters, clang-diagnostic-invalid-utf8, clang-diagnostic-invalid-source-encoding, clang-diagnostic-pointer-arith, clang-diagnostic-strict-prototypes, hicpp-uppercase-literal-suffix, cppcoreguidelines-*, performance-*)
```

#### BrbWcStringCountText.c - Zählt das Vorkommen einer Zeichenfolge innerhalb eines Texts
```c
/********************************************************************
 * COPYRIGHT -- Bernecker + Rainer
 ********************************************************************
 * Library: BrbLib
 * File: BrbWcStringCountText.c
 * Author: niedermeierr
 * Created: May 04, 2016
 ********************************************************************
 * Implementation of library BrbLib
 ********************************************************************/

#include <bur/plctypes.h>
#ifdef __cplusplus
	extern "C"
	{
#endif

#include "BrbLib.h"
#include <string.h>

#ifdef __cplusplus
	};
#endif

// NOLINTBEGIN(readability-*, bugprone-easily-swappable-parameters, clang-diagnostic-invalid-utf8, clang-diagnostic-invalid-source-encoding, clang-diagnostic-pointer-arith, clang-diagnostic-strict-prototypes, hicpp-uppercase-literal-suffix, cppcoreguidelines-*, performance-*)

/* Zählt das Vorkommen einer Zeichenfolge innerhalb eines Texts */
unsigned long BrbWcStringCountText(plcwstring* pText, plcwstring* pFind, unsigned long nTextLen)
{
	UDINT nResult = 0;
	// Wenn die Länge bekannt ist, kann sie übergeben werden
	// Damit entfällt das Aufrufen von strlen, welches bei langen Texten Zeit braucht
	UDINT nLenText = nTextLen;
	if(nTextLen == 0)
	{
		nLenText = brwcslen(pText);
	}
	UDINT nLenFind = brwcslen(pFind);
	UDINT nByteLenFind = nLenFind * 2;
	UDINT nCharIndex = 0;
	// Text von vorne nach hinten durchsuchen
	for(nCharIndex=0; nCharIndex<nLenText; nCharIndex++)
	{
		// Textstelle vergleichen
		if(memcmp((pText + nCharIndex), pFind, nByteLenFind) == 0)
		{
			// Text gefunden
			nResult += 1;
			nCharIndex += nLenFind-1;
		}
	}
	return nResult;
}

// NOLINTEND(readability-*, bugprone-easily-swappable-parameters, clang-diagnostic-invalid-utf8, clang-diagnostic-invalid-source-encoding, clang-diagnostic-pointer-arith, clang-diagnostic-strict-prototypes, hicpp-uppercase-literal-suffix, cppcoreguidelines-*, performance-*)
```

#### BrbWcStringRepeat.c - Wiederholt eine Zeichenfolge
```c
#include <bur/plctypes.h>
#ifdef __cplusplus
	extern "C"
	{
#endif

#include "BrbLib.h"
#include <string.h>

#ifdef __cplusplus
	};

#endif

// NOLINTBEGIN(readability-*, bugprone-easily-swappable-parameters, clang-diagnostic-invalid-utf8, clang-diagnostic-invalid-source-encoding, clang-diagnostic-pointer-arith, clang-diagnostic-strict-prototypes, hicpp-uppercase-literal-suffix, cppcoreguidelines-*, performance-*)

/* Wiederholt eine Zeichenfolge bis zu einer angegebenen Zeichenanzahl */
unsigned long BrbWcStringRepeat(plcwstring* pText, unsigned long nTextSize, plcwstring* pRepeat, unsigned long nLen)
{
	UDINT nCharCount = 0;
	UDINT nTextOffset = brwcslen(pText);
	UDINT nRepeatLen = brwcslen(pRepeat);
	// Länge limitieren
	if(nLen * 2 >= nTextSize)
	{
		nLen = (nTextSize-2)/2;
	}
	// Gesamten Wiederholtext wiederholend anhängen
	while(nTextOffset+nRepeatLen <= nLen)
	{
		BrbWcStringAppend(pText, pRepeat, &nTextOffset);
		nCharCount += nRepeatLen;
	}
	// Restliche Zeichen auffüllen
	DINT nCharCountLeft = (DINT)nLen - (DINT)nTextOffset;
	if(nCharCountLeft > 0)
	{
		UDINT nRepeatCharIndex = 0;
		for(nRepeatCharIndex=0; nRepeatCharIndex<(UDINT)nCharCountLeft; nRepeatCharIndex++)
		{
			//*(pText + nTextOffset) = *(pRepeat + nRepeatCharIndex);
			memcpy(pText + nTextOffset, pRepeat + nRepeatCharIndex, 2);
			nTextOffset++;
			nCharCount++;
		}
		*(pText + nTextOffset) = 0; // String-Abschluss
	}
	return nCharCount;
}

// NOLINTEND(readability-*, bugprone-easily-swappable-parameters, clang-diagnostic-invalid-utf8, clang-diagnostic-invalid-source-encoding, clang-diagnostic-pointer-arith, clang-diagnostic-strict-prototypes, hicpp-uppercase-literal-suffix, cppcoreguidelines-*, performance-*)
```
